C07210=1038.380,356.287,-127.366,172.660,43.947,158.571
C07211=1038.387,356.534,-127.405,172.666,43.949,158.572
C07212=1038.395,356.782,-127.444,172.672,43.953,158.573
C07213=1038.402,357.028,-127.482,172.677,43.955,158.575
C07214=1038.410,357.275,-127.521,172.684,43.958,158.576
C07215=1038.418,357.522,-127.559,172.690,43.962,158.577
C07216=1038.426,357.769,-127.598,172.695,43.965,158.578
C07217=1038.434,358.016,-127.636,172.702,43.968,158.580
C07218=1038.442,358.263,-127.674,172.708,43.971,158.581
C07219=1038.450,358.510,-127.713,172.714,43.974,158.582
C07220=1038.458,358.756,-127.751,172.720,43.978,158.584
C07221=1038.466,359.004,-127.790,172.727,43.981,158.585
C07222=1038.472,359.251,-127.829,172.732,43.983,158.586
C07223=1038.481,359.498,-127.867,172.738,43.987,158.587
C07224=1038.489,359.744,-127.907,172.744,43.990,158.589
C07225=1038.497,359.991,-127.945,172.750,43.993,158.590
C07226=1038.505,360.238,-127.984,172.757,43.996,158.591
C07227=1038.513,360.485,-128.022,172.763,44.000,158.593
C07228=1038.521,360.731,-128.061,172.769,44.003,158.594
C07229=1038.528,360.979,-128.100,172.775,44.006,158.595
C07230=1038.536,361.226,-128.139,172.782,44.009,158.597
C07231=1038.544,361.472,-128.178,172.787,44.013,158.598
C07232=1038.552,361.719,-128.216,172.794,44.016,158.599
C07233=1038.561,361.966,-128.256,172.800,44.019,158.601
C07234=1038.568,362.212,-128.295,172.807,44.022,158.602
C07235=1038.576,362.459,-128.334,172.812,44.026,158.603
C07236=1038.588,362.828,-128.393,172.822,44.031,158.605
C07237=1038.599,363.195,-128.451,172.832,44.036,158.608
C07238=1038.612,363.564,-128.509,172.840,44.041,158.610
C07239=1038.623,363.932,-128.568,172.850,44.046,158.612
C07240=1038.631,364.179,-128.607,172.857,44.049,158.613
C07241=1038.639,364.425,-128.646,172.862,44.052,158.614
C07242=1038.647,364.672,-128.686,172.869,44.056,158.616
C07243=1038.655,364.918,-128.725,172.875,44.059,158.617
C07244=1038.663,365.165,-128.765,172.882,44.063,158.619
C07245=1038.671,365.412,-128.804,172.888,44.067,158.620
C07246=1038.678,365.659,-128.844,172.894,44.070,158.621
C07247=1038.687,365.906,-128.883,172.901,44.073,158.623
C07248=1038.695,366.153,-128.923,172.907,44.077,158.624
C07249=1038.703,366.399,-128.962,172.914,44.080,158.626
C07250=1038.712,366.646,-129.002,172.921,44.083,158.627
C07251=1038.719,366.893,-129.041,172.927,44.087,158.629
C07252=1038.728,367.139,-129.081,172.934,44.091,158.630
C07253=1038.735,367.386,-129.121,172.940,44.094,158.632
C07254=1038.744,367.633,-129.160,172.946,44.098,158.633
C07255=1038.752,367.880,-129.200,172.953,44.101,158.634
C07256=1038.760,368.126,-129.239,172.960,44.105,158.636
C07257=1038.768,368.373,-129.280,172.966,44.109,158.637
C07258=1038.777,368.619,-129.319,172.973,44.112,158.639
C07259=1038.784,368.866,-129.359,172.980,44.115,158.640
C07260=1038.793,369.113,-129.399,172.986,44.119,158.642
C07261=1038.800,369.360,-129.438,172.993,44.123,158.643
C07262=1038.809,369.606,-129.478,172.999,44.126,158.645
C07263=1038.818,369.852,-129.518,173.006,44.130,158.646
C07264=1038.825,370.099,-129.558,173.012,44.134,158.648
C07265=1038.833,370.345,-129.598,173.019,44.137,158.649
C07266=1038.842,370.593,-129.638,173.026,44.141,158.651
C07267=1038.850,370.840,-129.678,173.033,44.145,158.652
C07268=1038.858,371.086,-129.719,173.039,44.149,158.654
C07269=1038.866,371.332,-129.759,173.046,44.152,158.655
C07270=1038.875,371.579,-129.799,173.053,44.156,158.657
C07271=1038.883,371.825,-129.839,173.060,44.159,158.658
C07272=1038.890,372.072,-129.879,173.066,44.163,158.660
C07273=1038.899,372.319,-129.920,173.073,44.168,158.662
C07274=1038.907,372.565,-129.961,173.080,44.171,158.663
C07275=1038.916,372.812,-130.000,173.087,44.175,158.665
C07276=1038.924,373.058,-130.041,173.094,44.179,158.666
C07277=1038.932,373.304,-130.081,173.100,44.182,158.668
C07278=1038.940,373.551,-130.122,173.108,44.187,158.669
C07279=1038.948,373.798,-130.162,173.115,44.190,158.671
C07280=1038.957,374.044,-130.202,173.121,44.194,158.672
C07281=1038.965,374.291,-130.243,173.128,44.198,158.674
C07282=1038.973,374.538,-130.284,173.136,44.202,158.676
C07283=1038.981,374.784,-130.325,173.143,44.206,158.677
C07284=1038.990,375.031,-130.366,173.150,44.210,158.679
C07285=1038.998,375.277,-130.406,173.156,44.214,158.680
C07286=1039.007,375.523,-130.446,173.163,44.217,158.682
C07287=1039.015,375.770,-130.487,173.170,44.221,158.684
C07288=1039.023,376.016,-130.528,173.177,44.225,158.685
C07289=1039.032,376.263,-130.569,173.184,44.229,158.687
C07290=1039.040,376.510,-130.610,173.191,44.233,158.688
C07291=1039.049,376.756,-130.650,173.199,44.237,158.690
C07292=1039.062,377.144,-130.714,173.210,44.244,158.693
C07293=1039.076,377.532,-130.778,173.221,44.250,158.695
C07294=1039.089,377.920,-130.843,173.233,44.256,158.698
C07295=1039.103,378.308,-130.908,173.244,44.263,158.701
C07296=1039.111,378.555,-130.949,173.251,44.266,158.702
C07297=1039.119,378.802,-130.989,173.259,44.270,158.704
C07298=1039.128,379.048,-131.031,173.266,44.275,158.706
C07299=1039.136,379.295,-131.072,173.273,44.279,158.707
C07300=1039.145,379.541,-131.114,173.280,44.283,158.709
C07301=1039.153,379.787,-131.155,173.288,44.287,158.711
C07302=1039.161,380.034,-131.196,173.295,44.291,158.712
C07303=1039.170,380.280,-131.238,173.302,44.296,158.714
C07304=1039.178,380.526,-131.279,173.309,44.300,158.716
C07305=1039.187,380.773,-131.321,173.317,44.304,158.718
C07306=1039.195,381.018,-131.362,173.324,44.308,158.719
C07307=1039.204,381.265,-131.403,173.331,44.312,158.721
C07308=1039.213,381.512,-131.445,173.339,44.317,158.723
C07309=1039.221,381.758,-131.486,173.346,44.321,158.725
C07310=1039.230,382.004,-131.528,173.354,44.325,158.726
C07311=1039.238,382.251,-131.570,173.361,44.329,158.728
C07312=1039.247,382.498,-131.611,173.369,44.334,158.730
C07313=1039.255,382.743,-131.653,173.376,44.338,158.732
C07314=1039.264,382.990,-131.695,173.383,44.343,158.733
C07315=1039.273,383.236,-131.736,173.391,44.347,158.735
C07316=1039.281,383.483,-131.779,173.399,44.351,158.737
C07317=1039.289,383.728,-131.820,173.406,44.355,158.739
C07318=1039.298,383.975,-131.862,173.414,44.360,158.741
C07319=1039.307,384.221,-131.903,173.421,44.364,158.742
C07320=1039.316,384.467,-131.945,173.429,44.369,158.744
C07321=1039.325,384.713,-131.988,173.437,44.373,158.746
C07322=1039.334,384.960,-132.030,173.445,44.378,158.748
C07323=1039.343,385.206,-132.072,173.452,44.382,158.750
C07324=1039.351,385.453,-132.113,173.460,44.387,158.752
C07325=1039.360,385.699,-132.155,173.468,44.391,158.754
C07326=1039.368,385.944,-132.198,173.475,44.395,158.755
C07327=1039.377,386.191,-132.239,173.483,44.400,158.757
C07328=1039.386,386.437,-132.281,173.491,44.405,158.759
C07329=1039.395,386.683,-132.323,173.498,44.409,158.761
C07330=1039.404,386.929,-132.366,173.506,44.414,158.763
C07331=1039.413,387.176,-132.408,173.515,44.418,158.765
C07332=1039.422,387.422,-132.450,173.522,44.423,158.767
C07333=1039.431,387.669,-132.492,173.531,44.427,158.769
C07334=1039.440,387.915,-132.535,173.538,44.432,158.770
C07335=1039.449,388.161,-132.577,173.546,44.437,158.772
C07336=1039.458,388.407,-132.619,173.554,44.441,158.774
C07337=1039.466,388.653,-132.662,173.562,44.446,158.776
C07338=1039.476,388.899,-132.705,173.570,44.450,158.778
C07339=1039.484,389.145,-132.747,173.578,44.455,158.780
C07340=1039.493,389.391,-132.789,173.585,44.460,158.782
C07341=1039.502,389.638,-132.833,173.594,44.464,158.784
C07342=1039.512,389.883,-132.875,173.601,44.469,158.786
C07343=1039.520,390.129,-132.918,173.610,44.474,158.788
C07344=1039.529,390.376,-132.960,173.618,44.479,158.790
C07345=1039.537,390.622,-133.003,173.626,44.483,158.792
C07346=1039.547,390.868,-133.046,173.634,44.489,158.794
C07347=1039.556,391.114,-133.089,173.643,44.493,158.796
C07348=1039.565,391.352,-133.130,173.650,44.498,158.798
C07349=1039.573,391.589,-133.172,173.658,44.502,158.800
C07350=1039.582,391.827,-133.214,173.666,44.507,158.802
C07351=1039.591,392.065,-133.255,173.674,44.512,158.804
C07352=1039.599,392.303,-133.297,173.682,44.517,158.806
C07353=1039.608,392.541,-133.338,173.690,44.521,158.808
C07354=1039.617,392.779,-133.380,173.698,44.526,158.809
C07355=1039.626,393.017,-133.422,173.707,44.531,158.812
C07356=1039.634,393.263,-133.465,173.714,44.536,158.813
C07357=1039.643,393.510,-133.508,173.723,44.541,158.816
C07358=1039.653,393.755,-133.551,173.732,44.546,158.818
C07359=1039.662,394.001,-133.595,173.740,44.551,158.820
C07360=1039.671,394.247,-133.638,173.748,44.555,158.822
C07361=1039.681,394.493,-133.681,173.756,44.561,158.824
C07362=1039.689,394.739,-133.725,173.765,44.566,158.826
C07363=1039.699,394.986,-133.768,173.774,44.571,158.828
C07364=1039.708,395.231,-133.812,173.783,44.576,158.830
C07365=1039.717,395.477,-133.855,173.790,44.581,158.832
C07366=1039.726,395.723,-133.899,173.799,44.586,158.834
C07367=1039.735,395.969,-133.943,173.808,44.591,158.837
C07368=1039.744,396.214,-133.987,173.816,44.596,158.839
C07369=1039.754,396.461,-134.029,173.825,44.602,158.841
C07370=1039.763,396.706,-134.073,173.834,44.607,158.843
C07371=1039.772,396.952,-134.117,173.843,44.612,158.845
C07372=1039.781,397.198,-134.161,173.851,44.617,158.847
C07373=1039.790,397.444,-134.205,173.860,44.623,158.850
C07374=1039.800,397.690,-134.249,173.868,44.628,158.852
C07375=1039.809,397.936,-134.293,173.877,44.632,158.854
C07376=1039.819,398.181,-134.336,173.886,44.638,158.856
C07377=1039.828,398.427,-134.381,173.894,44.643,158.858
C07378=1039.837,398.673,-134.424,173.903,44.649,158.861
C07379=1039.846,398.919,-134.468,173.912,44.654,158.863
C07380=1039.856,399.165,-134.512,173.921,44.659,158.865
C07381=1039.865,399.411,-134.557,173.930,44.664,158.867
C07382=1039.875,399.657,-134.601,173.939,44.670,158.870
C07383=1039.884,399.903,-134.646,173.948,44.675,158.872
C07384=1039.893,400.148,-134.689,173.957,44.680,158.874
C07385=1039.903,400.395,-134.733,173.966,44.686,158.876
C07386=1039.912,400.640,-134.778,173.975,44.691,158.879
C07387=1039.922,400.886,-134.822,173.985,44.697,158.881
C07388=1039.931,401.132,-134.867,173.994,44.702,158.883
C07389=1039.941,401.378,-134.911,174.003,44.708,158.886
C07390=1039.951,401.623,-134.956,174.012,44.714,158.888
C07391=1039.960,401.869,-135.000,174.021,44.719,158.890
C07392=1039.970,402.115,-135.045,174.030,44.725,158.893
C07393=1039.979,402.361,-135.090,174.039,44.730,158.895
C07394=1039.989,402.607,-135.134,174.049,44.736,158.897
C07395=1039.999,402.852,-135.179,174.058,44.741,158.900
C07396=1040.008,403.098,-135.224,174.067,44.747,158.902
C07397=1040.017,403.344,-135.268,174.076,44.753,158.905
C07398=1040.027,403.590,-135.313,174.085,44.758,158.907
C07399=1040.036,403.835,-135.358,174.094,44.764,158.909
C07400=1040.045,404.054,-135.398,174.103,44.769,158.911
C07401=1040.053,404.274,-135.439,174.111,44.774,158.914
C07402=1040.062,404.493,-135.479,174.119,44.779,158.916
C07403=1040.071,404.711,-135.519,174.128,44.784,158.918
C07404=1040.079,404.930,-135.559,174.136,44.789,158.920
C07405=1040.088,405.150,-135.600,174.145,44.794,158.922
C07406=1040.096,405.369,-135.640,174.153,44.800,158.924
C07407=1040.105,405.588,-135.681,174.162,44.805,158.927
C07408=1040.114,405.809,-135.721,174.171,44.810,158.929
C07409=1040.122,406.030,-135.762,174.179,44.816,158.931
C07410=1040.131,406.251,-135.802,174.188,44.820,158.933
C07411=1040.140,406.473,-135.843,174.196,44.826,158.936
C07412=1040.149,406.693,-135.883,174.205,44.831,158.938
C07413=1040.158,406.914,-135.925,174.214,44.837,158.940
C07414=1040.166,407.136,-135.966,174.222,44.842,158.942
C07415=1040.175,407.356,-136.006,174.231,44.847,158.945
C07416=1040.185,407.602,-136.053,174.241,44.853,158.947
C07417=1040.195,407.848,-136.098,174.251,44.859,158.950
C07418=1040.205,408.093,-136.144,174.261,44.865,158.952
C07419=1040.214,408.339,-136.189,174.271,44.871,158.955
C07420=1040.225,408.585,-136.235,174.280,44.877,158.957
C07421=1040.235,408.830,-136.280,174.290,44.883,158.960
C07422=1040.244,409.076,-136.326,174.301,44.889,158.963
C07423=1040.254,409.321,-136.372,174.310,44.895,158.965
C07424=1040.265,409.567,-136.417,174.321,44.901,158.968
C07425=1040.274,409.812,-136.463,174.330,44.907,158.970
C07426=1040.285,410.058,-136.509,174.341,44.913,158.973
C07427=1040.295,410.304,-136.555,174.350,44.920,158.976
C07428=1040.305,410.549,-136.601,174.361,44.925,158.978
C07429=1040.315,410.794,-136.647,174.371,44.932,158.981
C07430=1040.325,411.040,-136.693,174.381,44.938,158.984
C07431=1040.335,411.285,-136.739,174.391,44.944,158.986
C07432=1040.345,411.531,-136.785,174.401,44.950,158.989
C07433=1040.356,411.777,-136.831,174.412,44.957,158.992
C07434=1040.366,412.023,-136.878,174.422,44.963,158.994
C07435=1040.376,412.268,-136.924,174.432,44.969,158.997
C07436=1040.386,412.513,-136.971,174.442,44.976,159.000
C07437=1040.396,412.759,-137.017,174.453,44.982,159.003
C07438=1040.406,413.004,-137.063,174.464,44.988,159.005
C07439=1040.416,413.250,-137.110,174.473,44.995,159.008
C07440=1040.426,413.496,-137.157,174.484,45.001,159.011
C07441=1040.437,413.741,-137.204,174.495,45.008,159.014
C07442=1040.447,413.986,-137.250,174.506,45.014,159.017
C07443=1040.457,414.232,-137.297,174.516,45.020,159.019
C07444=1040.467,414.478,-137.344,174.527,45.027,159.022
C07445=1040.478,414.723,-137.390,174.537,45.034,159.025
C07446=1040.488,414.968,-137.437,174.548,45.040,159.028
C07447=1040.498,415.214,-137.484,174.558,45.047,159.031
C07448=1040.508,415.459,-137.531,174.569,45.053,159.033
C07449=1040.519,415.704,-137.578,174.580,45.060,159.036
C07450=1040.530,415.949,-137.625,174.591,45.067,159.039
C07451=1040.540,416.195,-137.672,174.602,45.073,159.042
C07452=1040.551,416.440,-137.719,174.613,45.080,159.045
C07453=1040.561,416.685,-137.766,174.624,45.086,159.048
C07454=1040.571,416.930,-137.813,174.635,45.093,159.051
C07455=1040.582,417.176,-137.861,174.646,45.099,159.054
C07456=1040.593,417.421,-137.907,174.657,45.106,159.057
C07457=1040.603,417.666,-137.955,174.668,45.113,159.060
C07458=1040.614,417.912,-138.002,174.679,45.120,159.063
C07459=1040.624,418.158,-138.049,174.690,45.127,159.066
C07460=1040.634,418.402,-138.097,174.701,45.134,159.069
C07461=1040.645,418.648,-138.145,174.712,45.141,159.072
C07462=1040.655,418.894,-138.192,174.723,45.147,159.075
C07463=1040.666,419.138,-138.240,174.735,45.154,159.078
C07464=1040.677,419.384,-138.288,174.746,45.161,159.081
C07465=1040.687,419.629,-138.336,174.757,45.168,159.084
C07466=1040.698,419.874,-138.384,174.769,45.175,159.087
C07467=1040.708,420.120,-138.431,174.780,45.182,159.090
C07468=1040.718,420.345,-138.475,174.790,45.189,159.093
C07469=1040.728,420.569,-138.519,174.801,45.195,159.096
C07470=1040.738,420.795,-138.563,174.812,45.201,159.099
C07471=1040.748,421.020,-138.607,174.822,45.208,159.102
C07472=1040.758,421.246,-138.651,174.833,45.214,159.104
C07473=1040.768,421.470,-138.696,174.844,45.221,159.107
C07474=1040.777,421.695,-138.739,174.855,45.227,159.110
C07475=1040.788,421.921,-138.784,174.865,45.234,159.113
C07476=1040.798,422.165,-138.832,174.877,45.241,159.116
C07477=1040.810,422.411,-138.881,174.889,45.248,159.119
C07478=1040.821,422.656,-138.929,174.900,45.255,159.123
C07479=1040.831,422.901,-138.977,174.913,45.262,159.126
C07480=1040.842,423.146,-139.025,174.924,45.270,159.129
C07481=1040.853,423.391,-139.073,174.937,45.277,159.132
C07482=1040.865,423.636,-139.122,174.948,45.284,159.136
C07483=1040.876,423.881,-139.171,174.961,45.292,159.139
C07484=1040.887,424.127,-139.219,174.972,45.299,159.142
C07485=1040.897,424.371,-139.268,174.985,45.307,159.146
C07486=1040.908,424.616,-139.317,174.997,45.314,159.149
C07487=1040.920,424.861,-139.366,175.009,45.321,159.152
C07488=1040.931,425.107,-139.414,175.021,45.329,159.156
C07489=1040.941,425.352,-139.463,175.033,45.336,159.159
C07490=1040.953,425.596,-139.512,175.046,45.344,159.162
C07491=1040.964,425.841,-139.561,175.058,45.351,159.166
C07492=1040.975,426.086,-139.610,175.070,45.359,159.169
C07493=1040.986,426.332,-139.659,175.083,45.366,159.172
C07494=1040.997,426.576,-139.708,175.095,45.374,159.176
C07495=1041.009,426.821,-139.757,175.108,45.381,159.179
C07496=1041.020,427.066,-139.806,175.120,45.389,159.183
C07497=1041.031,427.311,-139.856,175.133,45.397,159.186
C07498=1041.042,427.556,-139.905,175.146,45.404,159.190
C07499=1041.054,427.800,-139.954,175.158,45.412,159.193
C07500=1041.065,428.046,-140.004,175.171,45.420,159.197
C07501=1041.077,428.290,-140.054,175.184,45.427,159.200
C07502=1041.088,428.535,-140.103,175.197,45.435,159.204
C07503=1041.099,428.780,-140.152,175.210,45.443,159.207
C07504=1041.111,429.025,-140.202,175.223,45.451,159.211
C07505=1041.122,429.270,-140.252,175.236,45.458,159.214
C07506=1041.133,429.514,-140.302,175.249,45.466,159.218
C07507=1041.144,429.758,-140.352,175.262,45.474,159.222
C07508=1041.156,430.004,-140.401,175.275,45.482,159.225
C07509=1041.167,430.248,-140.452,175.288,45.490,159.229
C07510=1041.179,430.492,-140.502,175.301,45.498,159.232
C07511=1041.191,430.738,-140.552,175.314,45.506,159.236
C07512=1041.201,430.983,-140.602,175.327,45.515,159.240
C07513=1041.214,431.227,-140.652,175.340,45.523,159.243
C07514=1041.225,431.472,-140.702,175.354,45.530,159.247
C07515=1041.237,431.717,-140.752,175.368,45.539,159.251
C07516=1041.248,431.961,-140.803,175.381,45.547,159.255
C07517=1041.260,432.206,-140.853,175.394,45.555,159.258
C07518=1041.272,432.450,-140.904,175.408,45.563,159.262
C07519=1041.284,432.695,-140.954,175.421,45.571,159.266
C07520=1041.295,432.940,-141.005,175.435,45.579,159.270
C07521=1041.308,433.185,-141.055,175.449,45.588,159.274
C07522=1041.319,433.428,-141.106,175.463,45.596,159.277
C07523=1041.331,433.673,-141.156,175.477,45.604,159.281
C07524=1041.343,433.918,-141.207,175.490,45.613,159.285
C07525=1041.355,434.162,-141.257,175.505,45.621,159.289
C07526=1041.367,434.406,-141.308,175.518,45.629,159.293
C07527=1041.379,434.651,-141.358,175.532,45.637,159.297
C07528=1041.391,434.884,-141.407,175.546,45.646,159.301
C07529=1041.402,435.117,-141.456,175.559,45.653,159.304
C07530=1041.414,435.351,-141.504,175.572,45.662,159.308
C07531=1041.425,435.583,-141.553,175.586,45.669,159.312
C07532=1041.437,435.816,-141.602,175.600,45.678,159.316
C07533=1041.448,436.049,-141.650,175.613,45.686,159.319
C07534=1041.459,436.282,-141.700,175.628,45.694,159.323
C07535=1041.471,436.515,-141.749,175.641,45.702,159.327
C07536=1041.483,436.759,-141.800,175.656,45.711,159.331
C07537=1041.495,437.004,-141.851,175.670,45.720,159.335
C07538=1041.508,437.248,-141.903,175.684,45.728,159.339
C07539=1041.519,437.492,-141.955,175.699,45.737,159.344
C07540=1041.532,437.736,-142.006,175.714,45.746,159.348
C07541=1041.544,437.980,-142.058,175.728,45.754,159.352
C07542=1041.556,438.225,-142.109,175.743,45.763,159.356
C07543=1041.569,438.469,-142.162,175.758,45.772,159.360
C07544=1041.581,438.713,-142.214,175.773,45.781,159.364
C07545=1041.593,438.958,-142.265,175.788,45.789,159.368
C07546=1041.606,439.202,-142.318,175.803,45.799,159.373
C07547=1041.619,439.446,-142.369,175.818,45.808,159.377
C07548=1041.631,439.690,-142.421,175.833,45.817,159.381
C07549=1041.644,439.934,-142.474,175.849,45.825,159.386
C07550=1041.656,440.178,-142.526,175.864,45.834,159.390
C07551=1041.669,440.423,-142.578,175.879,45.844,159.394
C07552=1041.681,440.667,-142.630,175.894,45.853,159.399
C07553=1041.694,440.911,-142.683,175.910,45.861,159.403
C07554=1041.706,441.155,-142.735,175.925,45.871,159.407
C07555=1041.719,441.400,-142.788,175.941,45.880,159.412
C07556=1041.731,441.643,-142.840,175.957,45.889,159.416
C07557=1041.744,441.888,-142.893,175.972,45.898,159.421
C07558=1041.757,442.132,-142.946,175.988,45.907,159.425
C07559=1041.769,442.376,-142.998,176.004,45.917,159.430
C07560=1041.782,442.620,-143.051,176.020,45.926,159.434
C07561=1041.795,442.864,-143.104,176.035,45.935,159.439
C07562=1041.808,443.108,-143.157,176.052,45.944,159.443
C07563=1041.821,443.352,-143.210,176.067,45.954,159.448
C07564=1041.834,443.595,-143.263,176.084,45.964,159.452
C07565=1041.846,443.840,-143.316,176.100,45.973,159.457
C07566=1041.860,444.084,-143.369,176.116,45.982,159.461
C07567=1041.873,444.328,-143.422,176.132,45.992,159.466
C07568=1041.886,444.570,-143.475,176.149,46.001,159.471
C07569=1041.899,444.814,-143.528,176.165,46.011,159.476
C07570=1041.913,445.057,-143.581,176.182,46.020,159.480
C07571=1041.927,445.301,-143.634,176.199,46.030,159.485
C07572=1041.941,445.544,-143.686,176.215,46.039,159.489
C07573=1041.957,445.787,-143.737,176.231,46.048,159.494
C07574=1041.972,446.031,-143.788,176.248,46.057,159.499
C07575=1041.989,446.275,-143.839,176.265,46.066,159.503
C07576=1042.006,446.519,-143.889,176.282,46.075,159.508
C07577=1042.023,446.762,-143.939,176.299,46.083,159.512
C07578=1042.042,447.006,-143.988,176.316,46.092,159.517
C07579=1042.060,447.251,-144.037,176.333,46.100,159.521
C07580=1042.080,447.495,-144.084,176.351,46.109,159.526
C07581=1042.100,447.740,-144.132,176.368,46.117,159.530
C07582=1042.120,447.984,-144.180,176.385,46.125,159.535
C07583=1042.141,448.229,-144.226,176.402,46.133,159.539
C07584=1042.163,448.473,-144.273,176.420,46.141,159.544
C07585=1042.186,448.718,-144.319,176.439,46.149,159.548
C07586=1042.209,448.963,-144.364,176.455,46.157,159.552
C07587=1042.232,449.208,-144.408,176.473,46.165,159.557
C07588=1042.264,449.526,-144.466,176.497,46.174,159.562
C07589=1042.296,449.843,-144.523,176.520,46.184,159.568
C07590=1042.330,450.161,-144.579,176.543,46.193,159.573
C07591=1042.365,450.479,-144.633,176.567,46.202,159.579
C07592=1042.392,450.725,-144.676,176.586,46.209,159.583
C07593=1042.420,450.970,-144.717,176.603,46.216,159.587
C07594=1042.448,451.215,-144.758,176.622,46.223,159.592
C07595=1042.477,451.461,-144.799,176.641,46.230,159.596
C07596=1042.177,451.505,-145.113,176.644,46.308,159.620
C07597=1042.148,451.260,-145.073,176.625,46.302,159.616
C07598=1042.119,451.014,-145.032,176.606,46.295,159.611
C07599=1042.091,450.768,-144.991,176.588,46.289,159.607
C07600=1042.064,450.523,-144.949,176.570,46.281,159.603
C07601=1042.031,450.221,-144.897,176.546,46.273,159.598
C07602=1041.999,449.918,-144.844,176.524,46.264,159.592
C07603=1041.968,449.615,-144.790,176.502,46.255,159.587
C07604=1041.937,449.314,-144.736,176.480,46.246,159.582
C07605=1041.913,449.069,-144.692,176.462,46.238,159.577
C07606=1041.890,448.824,-144.646,176.444,46.231,159.573
C07607=1041.867,448.578,-144.600,176.427,46.223,159.568
C07608=1041.845,448.334,-144.555,176.409,46.215,159.564
C07609=1041.823,448.090,-144.508,176.391,46.207,159.560
C07610=1041.803,447.845,-144.461,176.373,46.199,159.555
C07611=1041.782,447.601,-144.414,176.356,46.191,159.551
C07612=1041.762,447.356,-144.366,176.339,46.183,159.546
C07613=1041.743,447.111,-144.317,176.321,46.174,159.542
C07614=1041.724,446.868,-144.268,176.304,46.166,159.537
C07615=1041.706,446.624,-144.219,176.287,46.157,159.533
C07616=1041.689,446.381,-144.169,176.270,46.149,159.528
C07617=1041.672,446.136,-144.118,176.253,46.140,159.524
C07618=1041.657,445.892,-144.068,176.236,46.131,159.519
C07619=1041.641,445.649,-144.016,176.219,46.122,159.514
C07620=1041.625,445.406,-143.965,176.203,46.113,159.510
C07621=1041.612,445.161,-143.913,176.186,46.104,159.505
C07622=1041.597,444.919,-143.860,176.170,46.095,159.501
C07623=1041.585,444.675,-143.807,176.153,46.085,159.496
C07624=1041.571,444.433,-143.755,176.137,46.076,159.491
C07625=1041.558,444.189,-143.701,176.120,46.067,159.487
C07626=1041.545,443.945,-143.648,176.103,46.057,159.482
C07627=1041.532,443.701,-143.595,176.088,46.048,159.477
C07628=1041.519,443.457,-143.542,176.072,46.038,159.473
C07629=1041.505,443.213,-143.489,176.055,46.029,159.468
C07630=1041.493,442.969,-143.436,176.040,46.020,159.464
C07631=1041.480,442.725,-143.383,176.023,46.011,159.459
C07632=1041.467,442.481,-143.330,176.007,46.001,159.455
C07633=1041.454,442.237,-143.277,175.992,45.992,159.450
C07634=1041.441,441.993,-143.224,175.975,45.983,159.446
C07635=1041.429,441.749,-143.172,175.960,45.974,159.441
C07636=1041.416,441.505,-143.119,175.944,45.965,159.437
C07637=1041.403,441.260,-143.066,175.928,45.955,159.432
C07638=1041.391,441.017,-143.014,175.913,45.946,159.428
C07639=1041.378,440.773,-142.961,175.897,45.938,159.424
C07640=1041.366,440.529,-142.909,175.882,45.929,159.419
C07641=1041.353,440.284,-142.857,175.867,45.920,159.415
C07642=1041.341,440.040,-142.804,175.851,45.911,159.411
C07643=1041.328,439.796,-142.752,175.836,45.902,159.406
C07644=1041.316,439.552,-142.700,175.821,45.893,159.402
C07645=1041.302,439.307,-142.648,175.806,45.884,159.398
C07646=1041.290,439.063,-142.597,175.791,45.875,159.393
C07647=1041.278,438.819,-142.544,175.775,45.866,159.389
C07648=1041.265,438.574,-142.492,175.760,45.858,159.385
C07649=1041.253,438.330,-142.441,175.745,45.849,159.381
C07650=1041.241,438.086,-142.388,175.730,45.840,159.377
C07651=1041.229,437.842,-142.337,175.715,45.832,159.373
C07652=1041.216,437.598,-142.285,175.700,45.823,159.368
C07653=1041.204,437.353,-142.234,175.686,45.814,159.364
C07654=1041.192,437.109,-142.182,175.672,45.805,159.360
C07655=1041.180,436.864,-142.130,175.657,45.797,159.356
C07656=1041.167,436.620,-142.079,175.643,45.789,159.352
C07657=1041.156,436.386,-142.030,175.628,45.781,159.348
C07658=1041.144,436.152,-141.981,175.615,45.772,159.344
C07659=1041.133,435.919,-141.932,175.601,45.764,159.340
C07660=1041.121,435.685,-141.883,175.587,45.756,159.336
C07661=1041.110,435.452,-141.834,175.574,45.748,159.333
C07662=1041.099,435.218,-141.785,175.560,45.740,159.329
C07663=1041.087,434.985,-141.736,175.546,45.732,159.325
C07664=1041.075,434.751,-141.688,175.533,45.724,159.321
C07665=1041.064,434.506,-141.637,175.518,45.716,159.317
C07666=1041.051,434.262,-141.586,175.505,45.707,159.314
C07667=1041.039,434.017,-141.535,175.491,45.699,159.310
C07668=1041.027,433.773,-141.485,175.477,45.691,159.306
C07669=1041.015,433.528,-141.434,175.463,45.683,159.302
C07670=1041.003,433.284,-141.383,175.449,45.674,159.298
C07671=1040.992,433.039,-141.333,175.435,45.666,159.294
C07672=1040.979,432.794,-141.283,175.422,45.658,159.290
C07673=1040.968,432.550,-141.232,175.407,45.650,159.287
C07674=1040.956,432.305,-141.181,175.394,45.642,159.283
C07675=1040.944,432.060,-141.131,175.381,45.634,159.279
C07676=1040.932,431.816,-141.081,175.367,45.626,159.275
C07677=1040.921,431.571,-141.030,175.353,45.618,159.272
C07678=1040.909,431.327,-140.981,175.340,45.609,159.268
C07679=1040.898,431.082,-140.930,175.327,45.601,159.264
C07680=1040.886,430.838,-140.880,175.313,45.594,159.260
C07681=1040.874,430.593,-140.830,175.300,45.586,159.257
C07682=1040.863,430.348,-140.780,175.287,45.578,159.253
C07683=1040.851,430.103,-140.730,175.274,45.570,159.250
C07684=1040.840,429.859,-140.680,175.261,45.562,159.246
C07685=1040.829,429.614,-140.630,175.248,45.554,159.242
C07686=1040.817,429.369,-140.580,175.235,45.546,159.239
C07687=1040.806,429.124,-140.530,175.221,45.538,159.235
C07688=1040.794,428.880,-140.480,175.209,45.531,159.232
C07689=1040.783,428.634,-140.430,175.196,45.523,159.228
C07690=1040.771,428.390,-140.381,175.183,45.516,159.224
C07691=1040.760,428.145,-140.331,175.170,45.508,159.221
C07692=1040.749,427.900,-140.282,175.157,45.500,159.217
C07693=1040.737,427.656,-140.233,175.144,45.492,159.214
C07694=1040.726,427.410,-140.183,175.131,45.485,159.210
C07695=1040.715,427.165,-140.134,175.119,45.477,159.207
C07696=1040.703,426.920,-140.085,175.106,45.470,159.203
C07697=1040.692,426.676,-140.036,175.093,45.462,159.200
C07698=1040.681,426.431,-139.986,175.081,45.455,159.197
C07699=1040.670,426.186,-139.937,175.069,45.447,159.193
C07700=1040.658,425.941,-139.888,175.056,45.440,159.190
C07701=1040.647,425.696,-139.839,175.043,45.432,159.186
C07702=1040.636,425.451,-139.790,175.031,45.425,159.183
C07703=1040.625,425.206,-139.741,175.019,45.417,159.180
C07704=1040.614,424.961,-139.692,175.006,45.410,159.176
C07705=1040.602,424.717,-139.643,174.995,45.402,159.173
C07706=1040.592,424.471,-139.595,174.982,45.396,159.170
C07707=1040.581,424.227,-139.546,174.969,45.388,159.166
C07708=1040.570,423.982,-139.498,174.958,45.381,159.163
C07709=1040.559,423.737,-139.449,174.945,45.373,159.160
C07710=1040.548,423.491,-139.400,174.934,45.366,159.156
C07711=1040.537,423.246,-139.352,174.921,45.359,159.153
C07712=1040.526,423.001,-139.304,174.910,45.352,159.150
C07713=1040.515,422.757,-139.255,174.898,45.345,159.147
C07714=1040.504,422.511,-139.207,174.886,45.338,159.144
C07715=1040.493,422.266,-139.158,174.874,45.331,159.140
C07716=1040.482,422.021,-139.110,174.862,45.324,159.137
C07717=1040.472,421.794,-139.065,174.851,45.317,159.134
C07718=1040.462,421.569,-139.021,174.840,45.310,159.131
C07719=1040.452,421.343,-138.977,174.830,45.304,159.128
C07720=1040.442,421.115,-138.933,174.819,45.297,159.125
C07721=1040.432,420.890,-138.889,174.808,45.291,159.123
C07722=1040.422,420.663,-138.844,174.797,45.284,159.120
C07723=1040.411,420.437,-138.800,174.787,45.278,159.117
C07724=1040.402,420.210,-138.756,174.776,45.272,159.114
C07725=1040.392,419.965,-138.708,174.765,45.264,159.111
C07726=1040.381,419.720,-138.659,174.753,45.258,159.108
C07727=1040.370,419.475,-138.612,174.742,45.251,159.105
C07728=1040.359,419.229,-138.564,174.730,45.244,159.102
C07729=1040.349,418.984,-138.517,174.719,45.237,159.099
C07730=1040.339,418.740,-138.469,174.708,45.231,159.096
C07731=1040.328,418.494,-138.421,174.697,45.223,159.093
C07732=1040.318,418.248,-138.374,174.686,45.217,159.090
C07733=1040.307,418.004,-138.326,174.674,45.210,159.087
C07734=1040.296,417.758,-138.278,174.663,45.203,159.084
C07735=1040.285,417.513,-138.232,174.652,45.197,159.081
C07736=1040.275,417.267,-138.185,174.640,45.190,159.078
C07737=1040.264,417.021,-138.137,174.630,45.184,159.075
C07738=1040.254,416.776,-138.090,174.619,45.177,159.072
C07739=1040.243,416.531,-138.043,174.607,45.170,159.069
C07740=1040.233,416.286,-137.996,174.597,45.164,159.066
C07741=1040.223,416.041,-137.949,174.586,45.157,159.063
C07742=1040.212,415.796,-137.902,174.575,45.150,159.060
C07743=1040.201,415.550,-137.854,174.565,45.144,159.057
C07744=1040.191,415.304,-137.807,174.554,45.137,159.054
C07745=1040.181,415.059,-137.760,174.543,45.131,159.052
C07746=1040.170,414.813,-137.714,174.532,45.125,159.049
C07747=1040.160,414.568,-137.667,174.521,45.118,159.046
C07748=1040.150,414.323,-137.620,174.510,45.112,159.043
C07749=1040.139,414.077,-137.574,174.499,45.105,159.040
C07750=1040.129,413.832,-137.527,174.490,45.099,159.038
C07751=1040.120,413.587,-137.480,174.479,45.093,159.035
C07752=1040.109,413.342,-137.434,174.468,45.086,159.032
C07753=1040.099,413.096,-137.387,174.457,45.079,159.029
C07754=1040.089,412.851,-137.340,174.447,45.073,159.026
C07755=1040.079,412.605,-137.294,174.437,45.067,159.024
C07756=1040.068,412.360,-137.247,174.426,45.061,159.021
C07757=1040.059,412.115,-137.201,174.416,45.054,159.018
C07758=1040.049,411.869,-137.154,174.406,45.048,159.015
C07759=1040.038,411.623,-137.108,174.395,45.042,159.013
C07760=1040.028,411.377,-137.062,174.385,45.036,159.010
C07761=1040.018,411.132,-137.016,174.374,45.030,159.007
C07762=1040.008,410.887,-136.970,174.365,45.023,159.005
C07763=1039.998,410.641,-136.924,174.354,45.017,159.002
C07764=1039.987,410.395,-136.878,174.344,45.011,158.999
C07765=1039.977,410.150,-136.832,174.334,45.005,158.997
C07766=1039.967,409.904,-136.786,174.324,44.999,158.994
C07767=1039.957,409.659,-136.740,174.314,44.993,158.991
C07768=1039.947,409.414,-136.695,174.303,44.987,158.989
C07769=1039.937,409.167,-136.649,174.294,44.981,158.986
C07770=1039.926,408.922,-136.603,174.283,44.975,158.984
C07771=1039.917,408.677,-136.557,174.274,44.969,158.981
C07772=1039.907,408.430,-136.512,174.263,44.963,158.978
C07773=1039.897,408.185,-136.466,174.254,44.957,158.976
C07774=1039.887,407.939,-136.420,174.244,44.951,158.973
C07775=1039.877,407.694,-136.375,174.234,44.945,158.971
C07776=1039.867,407.448,-136.330,174.224,44.939,158.968
C07777=1039.858,407.226,-136.288,174.215,44.934,158.966
C07778=1039.849,407.004,-136.247,174.206,44.929,158.964
C07779=1039.840,406.782,-136.206,174.198,44.924,158.962
C07780=1039.831,406.559,-136.165,174.189,44.918,158.959
C07781=1039.823,406.338,-136.124,174.180,44.913,158.957
C07782=1039.814,406.116,-136.083,174.172,44.908,158.955
C07783=1039.805,405.893,-136.042,174.163,44.902,158.952
C07784=1039.796,405.671,-136.001,174.154,44.897,158.950
C07785=1039.787,405.425,-135.955,174.144,44.891,158.948
C07786=1039.777,405.179,-135.911,174.135,44.886,158.945
C07787=1039.767,404.934,-135.866,174.126,44.880,158.943
C07788=1039.758,404.688,-135.820,174.116,44.875,158.940
C07789=1039.749,404.443,-135.775,174.106,44.869,158.938
C07790=1039.738,404.197,-135.730,174.097,44.863,158.936
C07791=1039.729,403.951,-135.685,174.088,44.858,158.933
C07792=1039.720,403.705,-135.640,174.078,44.852,158.931
C07793=1039.710,403.459,-135.595,174.069,44.846,158.928
C07794=1039.700,403.214,-135.550,174.060,44.841,158.926
C07795=1039.691,402.968,-135.505,174.050,44.835,158.924
C07796=1039.681,402.723,-135.460,174.041,44.829,158.921
C07797=1039.672,402.477,-135.416,174.031,44.824,158.919
C07798=1039.662,402.231,-135.371,174.022,44.818,158.916
C07799=1039.653,401.985,-135.326,174.013,44.813,158.914
C07800=1039.643,401.739,-135.282,174.004,44.807,158.912
C07801=1039.633,401.494,-135.237,173.995,44.802,158.909
C07802=1039.624,401.248,-135.193,173.986,44.797,158.907
C07803=1039.614,401.002,-135.149,173.977,44.791,158.905
C07804=1039.605,400.756,-135.104,173.968,44.786,158.903
C07805=1039.595,400.511,-135.060,173.958,44.780,158.900
C07806=1039.586,400.264,-135.016,173.949,44.775,158.898
C07807=1039.576,400.018,-134.971,173.940,44.770,158.896
C07808=1039.567,399.773,-134.927,173.931,44.764,158.893
C07809=1039.558,399.527,-134.883,173.922,44.759,158.891
C07810=1039.548,399.281,-134.839,173.913,44.754,158.889
C07811=1039.539,399.035,-134.795,173.904,44.748,158.887
C07812=1039.529,398.790,-134.750,173.895,44.743,158.884
C07813=1039.520,398.544,-134.706,173.886,44.738,158.882
C07814=1039.511,398.298,-134.662,173.878,44.733,158.880
C07815=1039.501,398.052,-134.618,173.869,44.728,158.878
C07816=1039.492,397.806,-134.574,173.861,44.723,158.876
C07817=1039.483,397.561,-134.531,173.851,44.717,158.873
C07818=1039.473,397.314,-134.486,173.843,44.712,158.871
C07819=1039.464,397.068,-134.442,173.834,44.707,158.869
C07820=1039.455,396.823,-134.399,173.826,44.702,158.867
C07821=1039.446,396.576,-134.355,173.817,44.696,158.865
C07822=1039.436,396.331,-134.312,173.808,44.691,158.862
C07823=1039.427,396.085,-134.268,173.799,44.686,158.860
C07824=1039.418,395.839,-134.224,173.790,44.681,158.858
C07825=1039.409,395.593,-134.181,173.782,44.676,158.856
C07826=1039.400,395.347,-134.137,173.773,44.671,158.854
C07827=1039.390,395.101,-134.094,173.765,44.666,158.852
C07828=1039.381,394.855,-134.050,173.757,44.661,158.850
C07829=1039.372,394.609,-134.006,173.748,44.656,158.848
C07830=1039.362,394.363,-133.964,173.739,44.651,158.846
C07831=1039.354,394.117,-133.920,173.730,44.646,158.843
C07832=1039.345,393.871,-133.877,173.723,44.641,158.841
C07833=1039.334,393.573,-133.824,173.712,44.635,158.839
C07834=1039.323,393.275,-133.772,173.702,44.629,158.836
C07835=1039.312,392.977,-133.720,173.691,44.623,158.834
C07836=1039.300,392.680,-133.667,173.681,44.618,158.831
C07837=1039.287,392.307,-133.602,173.669,44.611,158.828
C07838=1039.273,391.934,-133.536,173.657,44.603,158.825
C07839=1039.259,391.562,-133.472,173.644,44.596,158.822
C07840=1039.246,391.189,-133.407,173.632,44.588,158.819
C07841=1039.237,390.943,-133.364,173.623,44.584,158.817
C07842=1039.228,390.696,-133.320,173.616,44.579,158.815
C07843=1039.219,390.451,-133.278,173.607,44.574,158.813
C07844=1039.210,390.205,-133.235,173.599,44.569,158.811
C07845=1039.201,389.959,-133.192,173.591,44.565,158.809
C07846=1039.192,389.713,-133.151,173.583,44.560,158.807
C07847=1039.183,389.466,-133.107,173.575,44.556,158.805
C07848=1039.174,389.220,-133.065,173.567,44.551,158.803
C07849=1039.165,388.974,-133.022,173.559,44.547,158.801
C07850=1039.156,388.728,-132.979,173.551,44.541,158.799
C07851=1039.148,388.482,-132.937,173.542,44.537,158.797
C07852=1039.139,388.236,-132.895,173.535,44.533,158.796
C07853=1039.130,387.990,-132.852,173.526,44.528,158.794
C07854=1039.121,387.743,-132.810,173.519,44.523,158.792
C07855=1039.112,387.498,-132.767,173.511,44.519,158.790
C07856=1039.103,387.250,-132.725,173.503,44.514,158.788
C07857=1039.094,387.005,-132.682,173.495,44.510,158.786
C07858=1039.085,386.758,-132.641,173.487,44.506,158.784
C07859=1039.076,386.512,-132.599,173.479,44.501,158.782
C07860=1039.067,386.266,-132.556,173.472,44.496,158.780
C07861=1039.059,386.019,-132.514,173.463,44.492,158.779
C07862=1039.050,385.773,-132.472,173.456,44.488,158.777
C07863=1039.040,385.527,-132.430,173.448,44.483,158.775
C07864=1039.031,385.281,-132.388,173.440,44.479,158.773
C07865=1039.023,385.035,-132.347,173.432,44.474,158.771
C07866=1039.015,384.789,-132.305,173.425,44.470,158.769
C07867=1039.006,384.542,-132.263,173.418,44.466,158.768
C07868=1038.997,384.296,-132.221,173.409,44.461,158.766
C07869=1038.988,384.050,-132.179,173.402,44.457,158.764
C07870=1038.979,383.804,-132.137,173.394,44.452,158.762
C07871=1038.971,383.557,-132.095,173.386,44.449,158.760
C07872=1038.962,383.311,-132.053,173.379,44.444,158.759
C07873=1038.953,383.065,-132.012,173.371,44.440,158.757
C07874=1038.944,382.819,-131.970,173.364,44.435,158.755
C07875=1038.936,382.572,-131.928,173.357,44.431,158.753
C07876=1038.927,382.326,-131.886,173.348,44.427,158.751
C07877=1038.919,382.079,-131.845,173.341,44.423,158.750
C07878=1038.910,381.833,-131.804,173.334,44.418,158.748
C07879=1038.901,381.587,-131.762,173.326,44.414,158.746
C07880=1038.893,381.341,-131.721,173.319,44.410,158.744
C07881=1038.884,381.095,-131.679,173.312,44.406,158.743
C07882=1038.876,380.847,-131.637,173.305,44.402,158.741
C07883=1038.868,380.602,-131.596,173.296,44.398,158.739
C07884=1038.859,380.355,-131.554,173.289,44.394,158.737
C07885=1038.850,380.108,-131.513,173.282,44.389,158.736
C07886=1038.842,379.863,-131.472,173.274,44.385,158.734
C07887=1038.833,379.616,-131.431,173.267,44.381,158.732
C07888=1038.826,379.370,-131.389,173.260,44.377,158.731
C07889=1038.817,379.123,-131.347,173.253,44.373,158.729
C07890=1038.809,378.877,-131.307,173.245,44.368,158.727
C07891=1038.800,378.631,-131.265,173.238,44.365,158.726
C07892=1038.792,378.384,-131.224,173.231,44.361,158.724
C07893=1038.778,377.994,-131.159,173.220,44.354,158.721
C07894=1038.765,377.603,-131.094,173.208,44.348,158.718
C07895=1038.751,377.214,-131.030,173.197,44.342,158.716
C07896=1038.738,376.823,-130.965,173.185,44.335,158.713
C07897=1038.730,376.576,-130.925,173.178,44.332,158.712
C07898=1038.721,376.330,-130.883,173.171,44.327,158.710
C07899=1038.712,376.084,-130.843,173.164,44.324,158.708
C07900=1038.703,375.837,-130.802,173.157,44.320,158.707
C07901=1038.695,375.591,-130.761,173.150,44.316,158.705
C07902=1038.687,375.344,-130.720,173.143,44.312,158.704
C07903=1038.679,375.098,-130.680,173.135,44.308,158.702
C07904=1038.671,374.851,-130.639,173.128,44.304,158.700
C07905=1038.661,374.605,-130.599,173.121,44.301,158.699
C07906=1038.653,374.358,-130.558,173.114,44.297,158.697
C07907=1038.646,374.111,-130.518,173.107,44.293,158.696
C07908=1038.637,373.864,-130.477,173.101,44.289,158.694
C07909=1038.629,373.618,-130.436,173.094,44.285,158.693
C07910=1038.620,373.372,-130.396,173.087,44.282,158.691
C07911=1038.612,373.126,-130.356,173.080,44.278,158.689
C07912=1038.604,372.878,-130.315,173.073,44.274,158.688
C07913=1038.596,372.632,-130.275,173.066,44.270,158.686
C07914=1038.588,372.386,-130.234,173.059,44.267,158.685
C07915=1038.579,372.139,-130.195,173.053,44.263,158.683
C07916=1038.571,371.893,-130.154,173.046,44.259,158.682
C07917=1038.563,371.646,-130.113,173.039,44.255,158.680
C07918=1038.555,371.399,-130.073,173.032,44.252,158.679
C07919=1038.546,371.153,-130.033,173.025,44.248,158.677
C07920=1038.538,370.906,-129.993,173.019,44.244,158.675
C07921=1038.530,370.660,-129.953,173.012,44.241,158.674
C07922=1038.523,370.413,-129.913,173.005,44.237,158.672
C07923=1038.515,370.167,-129.872,172.998,44.233,158.671
C07924=1038.506,369.920,-129.833,172.992,44.229,158.669
C07925=1038.497,369.673,-129.793,172.985,44.226,158.668
C07926=1038.489,369.426,-129.752,172.978,44.223,158.666
C07927=1038.481,369.180,-129.713,172.971,44.219,158.665
C07928=1038.473,368.933,-129.673,172.964,44.215,158.663
C07929=1038.464,368.686,-129.634,172.959,44.212,158.662
C07930=1038.456,368.440,-129.593,172.952,44.208,158.661
C07931=1038.448,368.193,-129.554,172.945,44.205,158.659
C07932=1038.440,367.946,-129.514,172.939,44.201,158.658
C07933=1038.432,367.700,-129.475,172.932,44.198,158.656
C07934=1038.424,367.453,-129.435,172.925,44.195,158.655
C07935=1038.416,367.206,-129.395,172.918,44.191,158.653
C07936=1038.408,366.959,-129.355,172.912,44.188,158.652
C07937=1038.399,366.713,-129.316,172.905,44.184,158.650
C07938=1038.391,366.466,-129.277,172.899,44.181,158.649
C07939=1038.383,366.219,-129.237,172.893,44.177,158.647
C07940=1038.375,365.973,-129.198,172.886,44.174,158.646
C07941=1038.367,365.726,-129.158,172.880,44.171,158.645
C07942=1038.359,365.479,-129.118,172.873,44.167,158.643
C07943=1038.351,365.232,-129.078,172.867,44.164,158.642
C07944=1038.343,364.987,-129.039,172.861,44.160,158.640
C07945=1038.336,364.739,-129.000,172.854,44.157,158.639
C07946=1038.327,364.492,-128.961,172.847,44.154,158.638
C07947=1038.319,364.246,-128.922,172.841,44.150,158.636
C07948=1038.311,363.999,-128.882,172.834,44.147,158.635
C07949=1038.299,363.629,-128.823,172.825,44.142,158.633
C07950=1038.287,363.259,-128.764,172.816,44.137,158.631
C07951=1038.276,362.889,-128.706,172.807,44.132,158.629
C07952=1038.264,362.519,-128.647,172.797,44.127,158.627
C07953=1038.256,362.271,-128.608,172.790,44.124,158.625
C07954=1038.248,362.025,-128.568,172.784,44.120,158.624
C07955=1038.240,361.778,-128.530,172.778,44.117,158.623
C07956=1038.232,361.531,-128.490,172.772,44.114,158.621
C07957=1038.224,361.284,-128.451,172.765,44.111,158.620
C07958=1038.216,361.037,-128.413,172.760,44.108,158.619
C07959=1038.208,360.791,-128.374,172.753,44.104,158.617
C07960=1038.200,360.544,-128.335,172.747,44.101,158.616
C07961=1038.192,360.297,-128.297,172.740,44.098,158.615
C07962=1038.185,360.050,-128.257,172.735,44.095,158.613
C07963=1038.177,359.803,-128.218,172.728,44.091,158.612
C07964=1038.169,359.556,-128.180,172.722,44.089,158.611
C07965=1038.161,359.309,-128.142,172.716,44.086,158.609
C07966=1038.152,359.063,-128.102,172.710,44.082,158.608
C07967=1038.145,358.816,-128.064,172.704,44.079,158.607
C07968=1038.137,358.569,-128.025,172.698,44.076,158.606
C07969=1038.129,358.322,-127.987,172.692,44.073,158.604
C07970=1038.121,358.075,-127.949,172.685,44.070,158.603
C07971=1038.114,357.828,-127.909,172.680,44.067,158.602
C07972=1038.106,357.581,-127.871,172.673,44.064,158.600
C07973=1038.098,357.334,-127.833,172.667,44.061,158.599
C07974=1038.090,357.088,-127.794,172.662,44.058,158.598
C07975=1038.082,356.840,-127.756,172.655,44.055,158.597
C07976=1038.075,356.594,-127.717,172.650,44.051,158.595
C07977=1038.067,356.347,-127.679,172.644,44.049,158.594
C07978=1038.059,356.100,-127.641,172.637,44.046,158.593
C07979=1038.051,355.853,-127.602,172.632,44.043,158.592
C07980=1038.044,355.606,-127.564,172.625,44.040,158.590
C07981=1038.035,355.359,-127.526,172.620,44.037,158.589
C07982=1038.028,355.112,-127.488,172.614,44.034,158.588
C07983=1038.020,354.865,-127.449,172.608,44.031,158.587
C07984=1038.012,354.618,-127.412,172.602,44.028,158.585
C07985=1038.004,354.371,-127.374,172.596,44.025,158.584
C07986=1037.996,354.124,-127.335,172.590,44.022,158.583
C07987=1037.989,353.877,-127.298,172.584,44.020,158.582
C07988=1037.981,353.630,-127.259,172.579,44.016,158.581
C07989=1037.973,353.383,-127.221,172.572,44.014,158.579
C07990=1037.966,353.136,-127.183,172.567,44.011,158.578
C07991=1037.958,352.889,-127.145,172.561,44.008,158.577
C07992=1037.950,352.642,-127.108,172.555,44.005,158.576
C07993=1037.942,352.396,-127.070,172.549,44.002,158.575
C07994=1037.934,352.148,-127.032,172.544,43.999,158.573
C07995=1037.927,351.901,-126.993,172.538,43.996,158.572
C07996=1037.920,351.654,-126.956,172.532,43.994,158.571
C07997=1037.912,351.408,-126.918,172.526,43.991,158.570
C07998=1037.904,351.160,-126.880,172.521,43.988,158.569
C07999=1037.897,350.913,-126.842,172.515,43.985,158.567
C08000=1037.889,350.667,-126.805,172.509,43.983,158.566
C08001=1037.881,350.419,-126.767,172.503,43.980,158.565
C08002=1037.874,350.172,-126.729,172.498,43.977,158.564
C08003=1037.866,349.925,-126.691,172.492,43.974,158.563
C08004=1037.859,349.678,-126.653,172.487,43.971,158.562
C08005=1037.847,349.314,-126.598,172.478,43.968,158.560
C08006=1037.836,348.950,-126.543,172.470,43.963,158.558
C08007=1037.825,348.586,-126.488,172.461,43.959,158.557
C08008=1037.814,348.221,-126.432,172.453,43.955,158.555
C08009=1037.806,347.974,-126.395,172.448,43.953,158.554
C08010=1037.798,347.727,-126.358,172.442,43.950,158.553
C08011=1037.790,347.480,-126.321,172.436,43.948,158.552
C08012=1037.783,347.233,-126.283,172.431,43.945,158.550
C08013=1037.776,346.986,-126.246,172.425,43.942,158.549
C08014=1037.768,346.739,-126.209,172.420,43.939,158.548
C08015=1037.761,346.492,-126.171,172.415,43.937,158.547
C08016=1037.753,346.245,-126.134,172.409,43.934,158.546
C08017=1037.745,345.998,-126.097,172.403,43.932,158.545
C08018=1037.738,345.751,-126.059,172.397,43.929,158.544
C08019=1037.730,345.504,-126.022,172.392,43.927,158.543
C08020=1037.723,345.256,-125.985,172.387,43.924,158.542
C08021=1037.715,345.009,-125.948,172.381,43.921,158.540
C08022=1037.707,344.762,-125.911,172.376,43.919,158.539
C08023=1037.699,344.515,-125.874,172.370,43.916,158.538
C08024=1037.692,344.267,-125.837,172.365,43.914,158.537
C08025=1037.684,344.020,-125.800,172.360,43.911,158.536
C08026=1037.677,343.773,-125.763,172.354,43.908,158.535
C08027=1037.670,343.527,-125.726,172.348,43.906,158.534
C08028=1037.663,343.279,-125.689,172.343,43.903,158.533
C08029=1037.655,343.033,-125.652,172.337,43.901,158.532
C08030=1037.648,342.785,-125.616,172.332,43.898,158.531
C08031=1037.640,342.538,-125.579,172.327,43.896,158.530
C08032=1037.633,342.291,-125.541,172.321,43.893,158.529
C08033=1037.625,342.043,-125.505,172.316,43.891,158.528
C08034=1037.618,341.796,-125.467,172.311,43.888,158.527
C08035=1037.610,341.549,-125.431,172.305,43.886,158.526
C08036=1037.603,341.302,-125.394,172.300,43.883,158.525
C08037=1037.596,341.055,-125.358,172.295,43.881,158.524
C08038=1037.588,340.808,-125.322,172.290,43.879,158.523
C08039=1037.580,340.561,-125.285,172.284,43.876,158.521
C08040=1037.573,340.313,-125.248,172.279,43.874,158.520
C08041=1037.566,340.065,-125.212,172.274,43.872,158.519
C08042=1037.558,339.819,-125.175,172.269,43.870,158.519
C08043=1037.550,339.571,-125.138,172.263,43.867,158.517
C08044=1037.544,339.324,-125.102,172.258,43.865,158.516
C08045=1037.536,339.077,-125.066,172.253,43.862,158.515
C08046=1037.528,338.830,-125.029,172.248,43.860,158.514
C08047=1037.520,338.582,-124.993,172.242,43.857,158.513
C08048=1037.513,338.335,-124.956,172.237,43.855,158.512
C08049=1037.506,338.088,-124.920,172.232,43.853,158.511
C08050=1037.499,337.841,-124.884,172.226,43.851,158.510
C08051=1037.491,337.593,-124.847,172.221,43.848,158.509
C08052=1037.485,337.346,-124.811,172.216,43.846,158.508
C08053=1037.477,337.099,-124.774,172.211,43.843,158.507
C08054=1037.469,336.852,-124.738,172.205,43.841,158.506
C08055=1037.461,336.604,-124.702,172.200,43.839,158.505
C08056=1037.455,336.357,-124.665,172.196,43.837,158.504
C08057=1037.447,336.110,-124.629,172.191,43.834,158.504
C08058=1037.440,335.862,-124.593,172.186,43.832,158.503
C08059=1037.432,335.616,-124.557,172.180,43.830,158.502
C08060=1037.425,335.368,-124.521,172.175,43.828,158.501
C08061=1037.414,335.000,-124.467,172.168,43.825,158.499
C08062=1037.404,334.633,-124.414,172.160,43.821,158.498
C08063=1037.393,334.266,-124.360,172.153,43.818,158.496
C08064=1037.382,333.898,-124.306,172.145,43.815,158.495
C08065=1037.374,333.650,-124.271,172.140,43.813,158.494
C08066=1037.367,333.403,-124.236,172.135,43.810,158.493
C08067=1037.359,333.156,-124.199,172.130,43.808,158.492
C08068=1037.352,332.908,-124.164,172.124,43.806,158.491
C08069=1037.344,332.661,-124.128,172.120,43.803,158.490
C08070=1037.337,332.414,-124.092,172.115,43.802,158.489
C08071=1037.330,332.166,-124.057,172.110,43.800,158.488
C08072=1037.323,331.919,-124.021,172.105,43.797,158.488
C08073=1037.315,331.672,-123.985,172.100,43.795,158.487
C08074=1037.308,331.425,-123.949,172.095,43.793,158.486
C08075=1037.301,331.177,-123.913,172.090,43.791,158.485
C08076=1037.294,330.930,-123.878,172.085,43.789,158.484
C08077=1037.286,330.682,-123.842,172.080,43.787,158.483
C08078=1037.280,330.435,-123.807,172.075,43.785,158.482
C08079=1037.272,330.188,-123.770,172.070,43.783,158.481
C08080=1037.265,329.940,-123.735,172.065,43.780,158.480
C08081=1037.257,329.693,-123.699,172.061,43.779,158.479
C08082=1037.251,329.445,-123.664,172.056,43.776,158.478
C08083=1037.243,329.198,-123.628,172.051,43.774,158.477
C08084=1037.236,328.951,-123.593,172.046,43.773,158.477
C08085=1037.229,328.703,-123.558,172.041,43.770,158.476
C08086=1037.221,328.456,-123.522,172.036,43.768,158.475
C08087=1037.214,328.209,-123.487,172.031,43.766,158.474
C08088=1037.207,327.961,-123.451,172.026,43.765,158.473
C08089=1037.199,327.714,-123.417,172.021,43.762,158.472
C08090=1037.192,327.466,-123.381,172.017,43.761,158.471
C08091=1037.184,327.219,-123.346,172.012,43.758,158.470
C08092=1037.177,326.972,-123.311,172.007,43.757,158.470
C08093=1037.169,326.724,-123.276,172.002,43.755,158.469
C08094=1037.163,326.477,-123.241,171.998,43.753,158.468
C08095=1037.155,326.230,-123.206,171.993,43.751,158.467
C08096=1037.148,325.981,-123.171,171.988,43.749,158.466
C08097=1037.140,325.734,-123.136,171.983,43.747,158.465
C08098=1037.133,325.486,-123.101,171.979,43.745,158.465
C08099=1037.125,325.239,-123.066,171.974,43.744,158.464
C08100=1037.119,324.992,-123.031,171.969,43.741,158.463
C08101=1037.111,324.745,-122.996,171.964,43.740,158.462
C08102=1037.104,324.497,-122.961,171.960,43.738,158.461
C08103=1037.096,324.250,-122.926,171.955,43.736,158.461
C08104=1037.089,324.002,-122.891,171.950,43.734,158.460
C08105=1037.081,323.755,-122.856,171.946,43.732,158.459
C08106=1037.075,323.507,-122.821,171.941,43.730,158.458
C08107=1037.068,323.260,-122.786,171.936,43.729,158.457
C08108=1037.061,323.012,-122.752,171.931,43.727,158.456
C08109=1037.053,322.764,-122.717,171.927,43.725,158.455
C08110=1037.046,322.517,-122.682,171.922,43.723,158.455
C08111=1037.039,322.270,-122.647,171.917,43.721,158.454
C08112=1037.031,322.023,-122.613,171.913,43.720,158.453
C08113=1037.024,321.776,-122.578,171.908,43.717,158.452
C08114=1037.017,321.527,-122.543,171.903,43.716,158.451
C08115=1037.009,321.280,-122.509,171.899,43.714,158.451
C08116=1037.003,321.033,-122.474,171.894,43.712,158.450
C08117=1036.992,320.661,-122.421,171.887,43.709,158.449
C08118=1036.981,320.288,-122.369,171.880,43.707,158.447
C08119=1036.971,319.916,-122.317,171.873,43.704,158.446
C08120=1036.959,319.544,-122.265,171.866,43.701,158.445
C08121=1036.953,319.296,-122.231,171.862,43.699,158.444
C08122=1036.945,319.049,-122.196,171.857,43.698,158.443
C08123=1036.939,318.801,-122.161,171.853,43.696,158.443
C08124=1036.931,318.554,-122.127,171.848,43.694,158.442
C08125=1036.925,318.306,-122.092,171.843,43.693,158.441
C08126=1036.917,318.059,-122.058,171.839,43.691,158.440
C08127=1036.911,317.811,-122.023,171.834,43.689,158.439
C08128=1036.903,317.564,-121.990,171.830,43.687,158.439
C08129=1036.896,317.316,-121.955,171.825,43.686,158.438
C08130=1036.889,317.068,-121.921,171.820,43.684,158.437
C08131=1036.882,316.821,-121.886,171.816,43.682,158.436
C08132=1036.876,316.573,-121.852,171.811,43.680,158.436
C08133=1036.868,316.326,-121.818,171.807,43.678,158.435
C08134=1036.862,316.078,-121.783,171.802,43.677,158.434
C08135=1036.855,315.831,-121.749,171.799,43.675,158.433
C08136=1036.848,315.584,-121.714,171.794,43.673,158.432
C08137=1036.841,315.336,-121.680,171.790,43.672,158.432
C08138=1036.834,315.089,-121.646,171.785,43.670,158.431
C08139=1036.827,314.841,-121.611,171.781,43.669,158.430
C08140=1036.820,314.594,-121.577,171.776,43.667,158.429
C08141=1036.813,314.346,-121.543,171.772,43.665,158.429
C08142=1036.806,314.098,-121.509,171.767,43.663,158.428
C08143=1036.800,313.851,-121.474,171.763,43.661,158.427
C08144=1036.793,313.604,-121.441,171.758,43.660,158.426
C08145=1036.786,313.356,-121.407,171.755,43.659,158.426
C08146=1036.779,313.108,-121.372,171.750,43.657,158.425
C08147=1036.772,312.861,-121.338,171.746,43.655,158.424
C08148=1036.766,312.614,-121.304,171.741,43.653,158.423
C08149=1036.759,312.366,-121.270,171.737,43.651,158.423
C08150=1036.751,312.118,-121.236,171.732,43.650,158.422
C08151=1036.745,311.870,-121.202,171.728,43.649,158.421
C08152=1036.738,311.623,-121.168,171.723,43.647,158.420
C08153=1036.730,311.375,-121.134,171.719,43.646,158.420
C08154=1036.724,311.128,-121.101,171.714,43.644,158.419
C08155=1036.716,310.881,-121.067,171.711,43.642,158.418
C08156=1036.709,310.633,-121.034,171.706,43.641,158.418
C08157=1036.702,310.385,-121.000,171.702,43.639,158.417
C08158=1036.694,310.138,-120.966,171.697,43.638,158.416
C08159=1036.687,309.889,-120.933,171.693,43.636,158.416
C08160=1036.681,309.642,-120.899,171.689,43.635,158.415
C08161=1036.673,309.395,-120.866,171.685,43.633,158.414
C08162=1036.666,309.147,-120.832,171.680,43.632,158.414
C08163=1036.659,308.900,-120.798,171.676,43.631,158.413
C08164=1036.652,308.652,-120.766,171.672,43.629,158.412
C08165=1036.645,308.404,-120.732,171.667,43.628,158.412
C08166=1036.637,308.157,-120.699,171.664,43.626,158.411
C08167=1036.630,307.909,-120.666,171.659,43.625,158.410
C08168=1036.624,307.662,-120.632,171.655,43.623,158.409
C08169=1036.616,307.414,-120.598,171.650,43.622,158.409
C08170=1036.609,307.166,-120.564,171.646,43.621,158.408
C08171=1036.602,306.918,-120.531,171.642,43.619,158.407
C08172=1036.595,306.671,-120.498,171.638,43.618,158.407
C08173=1036.585,306.304,-120.449,171.632,43.616,158.406
C08174=1036.574,305.936,-120.399,171.625,43.614,158.405
C08175=1036.563,305.569,-120.350,171.619,43.612,158.404
C08176=1036.553,305.201,-120.301,171.613,43.610,158.403
C08177=1036.547,304.954,-120.268,171.608,43.608,158.402
C08178=1036.540,304.706,-120.234,171.604,43.607,158.401
C08179=1036.533,304.459,-120.202,171.601,43.605,158.401
C08180=1036.525,304.211,-120.168,171.596,43.604,158.400
C08181=1036.518,303.963,-120.135,171.592,43.602,158.399
C08182=1036.512,303.716,-120.101,171.587,43.601,158.399
C08183=1036.505,303.468,-120.068,171.584,43.600,158.398
C08184=1036.498,303.221,-120.035,171.580,43.598,158.397
C08185=1036.491,302.973,-120.002,171.575,43.597,158.397
C08186=1036.484,302.725,-119.970,171.571,43.596,158.396
C08187=1036.477,302.477,-119.936,171.568,43.595,158.396
C08188=1036.470,302.230,-119.904,171.563,43.593,158.395
C08189=1036.463,301.982,-119.871,171.559,43.592,158.394
C08190=1036.457,301.735,-119.837,171.555,43.590,158.394
C08191=1036.450,301.487,-119.804,171.551,43.589,158.393
C08192=1036.444,301.239,-119.771,171.547,43.587,158.392
C08193=1036.436,300.992,-119.738,171.543,43.586,158.392
C08194=1036.429,300.744,-119.705,171.538,43.585,158.391
C08195=1036.422,300.496,-119.672,171.534,43.584,158.390
C08196=1036.416,300.248,-119.639,171.531,43.582,158.390
C08197=1036.408,300.001,-119.606,171.526,43.581,158.389
C08198=1036.402,299.753,-119.573,171.522,43.579,158.388
C08199=1036.395,299.505,-119.540,171.518,43.578,158.388
C08200=1036.389,299.257,-119.508,171.515,43.577,158.387
C08201=1036.382,299.010,-119.475,171.510,43.576,158.387
C08202=1036.374,298.762,-119.442,171.506,43.574,158.386
C08203=1036.368,298.515,-119.409,171.502,43.573,158.385
C08204=1036.361,298.266,-119.376,171.499,43.571,158.385
C08205=1036.354,298.019,-119.344,171.494,43.570,158.384
C08206=1036.348,297.772,-119.311,171.490,43.569,158.384
C08207=1036.341,297.523,-119.278,171.486,43.568,158.383
C08208=1036.335,297.276,-119.245,171.483,43.567,158.382
C08209=1036.328,297.028,-119.213,171.478,43.565,158.382
C08210=1036.321,296.780,-119.180,171.474,43.564,158.381
C08211=1036.315,296.532,-119.147,171.470,43.562,158.380
C08212=1036.308,296.285,-119.114,171.467,43.561,158.380
C08213=1036.301,296.037,-119.082,171.462,43.560,158.379
C08214=1036.294,295.789,-119.049,171.458,43.559,158.379
C08215=1036.288,295.542,-119.016,171.455,43.557,158.378
C08216=1036.280,295.294,-118.984,171.451,43.556,158.377
C08217=1036.274,295.046,-118.951,171.447,43.555,158.377
C08218=1036.268,294.799,-118.918,171.442,43.554,158.376
C08219=1036.260,294.551,-118.886,171.439,43.552,158.376
C08220=1036.253,294.303,-118.854,171.435,43.551,158.375
C08221=1036.247,294.055,-118.822,171.431,43.550,158.374
C08222=1036.240,293.807,-118.789,171.427,43.549,158.374
C08223=1036.233,293.559,-118.756,171.423,43.548,158.373
C08224=1036.226,293.312,-118.724,171.419,43.547,158.373
C08225=1036.220,293.064,-118.692,171.416,43.546,158.372
C08226=1036.213,292.816,-118.660,171.412,43.544,158.372
C08227=1036.206,292.569,-118.627,171.407,43.543,158.371
C08228=1036.199,292.321,-118.596,171.404,43.542,158.370
C08229=1036.189,291.970,-118.550,171.399,43.540,158.369
C08230=1036.180,291.619,-118.505,171.393,43.539,158.369
C08231=1036.170,291.269,-118.459,171.388,43.537,158.368
C08232=1036.161,290.918,-118.414,171.382,43.535,158.367
C08233=1036.153,290.670,-118.381,171.378,43.535,158.367
C08234=1036.146,290.422,-118.350,171.375,43.533,158.366
C08235=1036.140,290.175,-118.317,171.371,43.532,158.365
C08236=1036.133,289.927,-118.286,171.366,43.531,158.365
C08237=1036.126,289.679,-118.253,171.363,43.530,158.364
C08238=1036.119,289.431,-118.222,171.359,43.529,158.364
C08239=1036.113,289.183,-118.189,171.355,43.528,158.363
C08240=1036.106,288.935,-118.158,171.352,43.527,158.363
C08241=1036.099,288.688,-118.125,171.348,43.526,158.362
C08242=1036.092,288.440,-118.094,171.344,43.525,158.362
C08243=1036.085,288.192,-118.062,171.340,43.524,158.361
C08244=1036.079,287.944,-118.029,171.336,43.523,158.361
C08245=1036.072,287.696,-117.998,171.333,43.522,158.360
C08246=1036.065,287.449,-117.966,171.329,43.520,158.359
C08247=1036.058,287.201,-117.934,171.325,43.520,158.359
C08248=1036.051,286.953,-117.903,171.322,43.518,158.358
C08249=1036.045,286.705,-117.871,171.317,43.517,158.358
C08250=1036.038,286.457,-117.838,171.314,43.517,158.357
C08251=1036.031,286.209,-117.807,171.310,43.515,158.357
C08252=1036.024,285.961,-117.776,171.306,43.515,158.356
C08253=1036.018,285.713,-117.744,171.303,43.513,158.356
C08254=1036.011,285.466,-117.712,171.299,43.513,158.355
C08255=1036.004,285.218,-117.681,171.295,43.511,158.355
C08256=1035.997,284.970,-117.649,171.292,43.511,158.354
C08257=1035.990,284.721,-117.617,171.287,43.510,158.354
C08258=1035.983,284.474,-117.586,171.284,43.509,158.353
C08259=1035.976,284.226,-117.554,171.280,43.508,158.353
C08260=1035.969,283.978,-117.524,171.277,43.507,158.352
C08261=1035.962,283.730,-117.492,171.273,43.506,158.351
C08262=1035.955,283.482,-117.461,171.269,43.505,158.351
C08263=1035.948,283.235,-117.429,171.266,43.504,158.350
C08264=1035.942,282.987,-117.397,171.262,43.503,158.350
C08265=1035.935,282.739,-117.366,171.259,43.502,158.349
C08266=1035.928,282.491,-117.334,171.255,43.501,158.349
C08267=1035.921,282.243,-117.303,171.251,43.500,158.348
C08268=1035.915,281.995,-117.271,171.248,43.499,158.348
C08269=1035.908,281.748,-117.240,171.243,43.498,158.347
C08270=1035.901,281.500,-117.209,171.240,43.497,158.347
C08271=1035.895,281.252,-117.177,171.236,43.496,158.346
C08272=1035.888,281.003,-117.146,171.233,43.495,158.346
C08273=1035.881,280.755,-117.115,171.229,43.494,158.345
C08274=1035.875,280.507,-117.084,171.225,43.493,158.345
C08275=1035.868,280.260,-117.052,171.222,43.492,158.344
C08276=1035.861,280.012,-117.021,171.218,43.491,158.344
C08277=1035.854,279.764,-116.989,171.215,43.491,158.343
C08278=1035.848,279.516,-116.958,171.211,43.489,158.343
C08279=1035.841,279.268,-116.926,171.208,43.489,158.342
C08280=1035.834,279.020,-116.895,171.204,43.487,158.342
C08281=1035.828,278.772,-116.864,171.200,43.487,158.341
C08282=1035.821,278.524,-116.833,171.197,43.486,158.341
C08283=1035.814,278.276,-116.802,171.193,43.485,158.340
C08284=1035.808,278.029,-116.771,171.190,43.484,158.340
C08285=1035.798,277.689,-116.729,171.185,43.483,158.339
C08286=1035.789,277.351,-116.686,171.180,43.482,158.339
C08287=1035.780,277.012,-116.644,171.175,43.480,158.338
C08288=1035.770,276.673,-116.602,171.171,43.479,158.337
C08289=1035.764,276.426,-116.570,171.167,43.478,158.337
C08290=1035.757,276.177,-116.540,171.164,43.478,158.336
C08291=1035.750,275.929,-116.509,171.160,43.477,158.336
C08292=1035.743,275.682,-116.477,171.157,43.476,158.335
C08293=1035.737,275.434,-116.447,171.153,43.475,158.335
C08294=1035.730,275.186,-116.416,171.150,43.474,158.334
C08295=1035.723,274.938,-116.385,171.146,43.474,158.334
C08296=1035.717,274.690,-116.354,171.142,43.472,158.333
C08297=1035.710,274.441,-116.323,171.139,43.472,158.333
C08298=1035.703,274.194,-116.293,171.135,43.471,158.333
C08299=1035.697,273.946,-116.262,171.132,43.470,158.332
C08300=1035.689,273.698,-116.231,171.128,43.469,158.332
C08301=1035.683,273.450,-116.201,171.125,43.468,158.331
C08302=1035.676,273.202,-116.169,171.121,43.468,158.331
C08303=1035.669,272.954,-116.139,171.118,43.467,158.330
C08304=1035.662,272.706,-116.108,171.114,43.466,158.330
C08305=1035.657,272.458,-116.077,171.111,43.466,158.329
C08306=1035.649,272.210,-116.047,171.107,43.464,158.329
C08307=1035.643,271.962,-116.016,171.104,43.464,158.328
C08308=1035.636,271.714,-115.986,171.100,43.463,158.328
C08309=1035.629,271.466,-115.954,171.097,43.462,158.328
C08310=1035.623,271.218,-115.924,171.093,43.462,158.327
C08311=1035.616,270.970,-115.894,171.090,43.461,158.327
C08312=1035.609,270.721,-115.863,171.086,43.460,158.326
C08313=1035.602,270.473,-115.832,171.084,43.459,158.326
C08314=1035.596,270.226,-115.802,171.080,43.458,158.325
C08315=1035.589,269.977,-115.772,171.077,43.457,158.325
C08316=1035.582,269.729,-115.742,171.073,43.457,158.324
C08317=1035.575,269.481,-115.710,171.070,43.456,158.324
C08318=1035.569,269.234,-115.680,171.066,43.455,158.324
C08319=1035.562,268.985,-115.650,171.063,43.455,158.323
C08320=1035.555,268.737,-115.620,171.059,43.454,158.323
C08321=1035.549,268.489,-115.589,171.056,43.453,158.322
C08322=1035.542,268.242,-115.558,171.052,43.453,158.322
C08323=1035.535,267.993,-115.528,171.049,43.452,158.321
C08324=1035.528,267.745,-115.497,171.046,43.451,158.321
C08325=1035.522,267.497,-115.468,171.043,43.450,158.321
C08326=1035.515,267.249,-115.437,171.040,43.450,158.320
C08327=1035.508,267.001,-115.407,171.036,43.449,158.320
C08328=1035.502,266.753,-115.377,171.033,43.448,158.319
C08329=1035.495,266.505,-115.346,171.029,43.448,158.319
C08330=1035.488,266.256,-115.316,171.026,43.447,158.318
C08331=1035.481,266.009,-115.287,171.022,43.446,158.318
C08332=1035.475,265.760,-115.256,171.019,43.445,158.318
C08333=1035.468,265.512,-115.226,171.016,43.445,158.317
C08334=1035.461,265.265,-115.196,171.013,43.444,158.317
C08335=1035.455,265.016,-115.165,171.009,43.443,158.316
C08336=1035.448,264.768,-115.135,171.006,43.442,158.316
C08337=1035.441,264.520,-115.105,171.002,43.442,158.315
C08338=1035.434,264.272,-115.075,170.999,43.441,158.315
C08339=1035.427,264.024,-115.045,170.995,43.440,158.315
C08340=1035.421,263.776,-115.015,170.993,43.440,158.314
C08341=1035.412,263.442,-114.974,170.988,43.439,158.314
C08342=1035.403,263.108,-114.934,170.984,43.438,158.313
C08343=1035.394,262.774,-114.893,170.979,43.437,158.313
C08344=1035.385,262.440,-114.853,170.975,43.436,158.312
C08345=1035.378,262.191,-114.823,170.971,43.436,158.312
C08346=1035.372,261.944,-114.793,170.969,43.435,158.311
C08347=1035.365,261.695,-114.764,170.965,43.434,158.311
C08348=1035.358,261.447,-114.734,170.962,43.434,158.310
C08349=1035.351,261.199,-114.704,170.958,43.433,158.310
C08350=1035.344,260.950,-114.674,170.955,43.433,158.310
C08351=1035.338,260.703,-114.645,170.951,43.432,158.309
C08352=1035.330,260.455,-114.614,170.949,43.432,158.309
C08353=1035.324,260.207,-114.585,170.946,43.431,158.308
C08354=1035.317,259.958,-114.555,170.942,43.430,158.308
C08355=1035.310,259.710,-114.526,170.939,43.430,158.308
C08356=1035.303,259.462,-114.497,170.936,43.429,158.307
C08357=1035.296,259.214,-114.467,170.932,43.429,158.307
C08358=1035.290,258.966,-114.438,170.930,43.429,158.307
C08359=1035.282,258.718,-114.407,170.926,43.428,158.306
C08360=1035.276,258.469,-114.378,170.923,43.427,158.306
C08361=1035.269,258.221,-114.348,170.919,43.426,158.305
C08362=1035.262,257.973,-114.319,170.916,43.426,158.305
C08363=1035.256,257.725,-114.289,170.913,43.426,158.305
C08364=1035.249,257.476,-114.260,170.910,43.425,158.304
C08365=1035.241,257.229,-114.231,170.907,43.425,158.304
C08366=1035.235,256.980,-114.201,170.903,43.424,158.304
C08367=1035.228,256.732,-114.172,170.900,43.423,158.303
C08368=1035.221,256.484,-114.142,170.897,43.423,158.303
C08369=1035.215,256.236,-114.113,170.894,43.422,158.302
C08370=1035.208,255.988,-114.083,170.891,43.422,158.302
C08371=1035.202,255.739,-114.054,170.888,43.422,158.302
C08372=1035.194,255.491,-114.024,170.884,43.421,158.301
C08373=1035.187,255.243,-113.995,170.882,43.420,158.301
C08374=1035.181,254.995,-113.966,170.878,43.420,158.301
C08375=1035.174,254.747,-113.936,170.875,43.419,158.300
C08376=1035.167,254.498,-113.907,170.871,43.419,158.300
C08377=1035.161,254.250,-113.878,170.869,43.418,158.300
C08378=1035.154,254.003,-113.848,170.866,43.418,158.299
C08379=1035.147,253.754,-113.818,170.862,43.417,158.299
C08380=1035.140,253.506,-113.790,170.859,43.417,158.298
C08381=1035.133,253.258,-113.760,170.857,43.416,158.298
C08382=1035.127,253.010,-113.731,170.853,43.415,158.298
C08383=1035.121,252.761,-113.702,170.850,43.415,158.297
C08384=1035.114,252.513,-113.672,170.846,43.414,158.297
C08385=1035.107,252.265,-113.643,170.844,43.414,158.297
C08386=1035.100,252.017,-113.614,170.841,43.414,158.296
C08387=1035.094,251.768,-113.585,170.837,43.413,158.296
C08388=1035.087,251.520,-113.556,170.834,43.413,158.295
C08389=1035.080,251.271,-113.526,170.831,43.412,158.295
C08390=1035.074,251.024,-113.497,170.828,43.411,158.295
C08391=1035.068,250.776,-113.468,170.825,43.411,158.294
C08392=1035.061,250.527,-113.438,170.822,43.410,158.294
C08393=1035.054,250.279,-113.410,170.819,43.410,158.294
C08394=1035.048,250.031,-113.381,170.815,43.409,158.293
C08395=1035.041,249.782,-113.351,170.813,43.409,158.293
C08396=1035.034,249.535,-113.321,170.810,43.408,158.293
C08397=1035.025,249.199,-113.282,170.805,43.408,158.292
C08398=1035.016,248.863,-113.244,170.802,43.407,158.292
C08399=1035.007,248.528,-113.204,170.797,43.406,158.291
C08400=1034.999,248.193,-113.165,170.794,43.405,158.291
C08401=1034.993,247.944,-113.135,170.790,43.405,158.290
C08402=1034.985,247.696,-113.107,170.787,43.405,158.290
C08403=1034.979,247.448,-113.078,170.784,43.404,158.290
C08404=1034.972,247.200,-113.049,170.781,43.404,158.289
C08405=1034.966,246.951,-113.020,170.778,43.403,158.289
C08406=1034.959,246.703,-112.990,170.775,43.403,158.289
C08407=1034.953,246.455,-112.961,170.772,43.402,158.288
C08408=1034.946,246.207,-112.933,170.769,43.401,158.288
C08409=1034.940,245.959,-112.904,170.766,43.401,158.288
C08410=1034.934,245.710,-112.875,170.763,43.400,158.287
C08411=1034.927,245.462,-112.845,170.761,43.400,158.287
C08412=1034.921,245.213,-112.816,170.757,43.399,158.286
C08413=1034.914,244.966,-112.788,170.754,43.399,158.286
C08414=1034.907,244.718,-112.759,170.751,43.398,158.286
C08415=1034.901,244.469,-112.730,170.748,43.398,158.285
C08416=1034.893,244.221,-112.701,170.745,43.398,158.285
C08417=1034.887,243.973,-112.672,170.742,43.397,158.285
C08418=1034.881,243.724,-112.644,170.739,43.397,158.284
C08419=1034.874,243.476,-112.615,170.737,43.396,158.284
C08420=1034.867,243.228,-112.586,170.733,43.396,158.284
C08421=1034.860,242.980,-112.557,170.730,43.396,158.283
C08422=1034.855,242.731,-112.529,170.728,43.395,158.283
C08423=1034.848,242.483,-112.500,170.724,43.395,158.283
C08424=1034.841,242.235,-112.471,170.721,43.394,158.282
C08425=1034.834,241.986,-112.443,170.719,43.394,158.282
C08426=1034.828,241.738,-112.414,170.715,43.393,158.282
C08427=1034.821,241.490,-112.386,170.713,43.393,158.281
C08428=1034.815,241.242,-112.357,170.710,43.393,158.281
C08429=1034.808,240.993,-112.329,170.706,43.392,158.281
C08430=1034.802,240.745,-112.300,170.704,43.392,158.280
C08431=1034.795,240.497,-112.271,170.700,43.391,158.280
C08432=1034.788,240.248,-112.243,170.698,43.391,158.280
C08433=1034.781,240.000,-112.214,170.695,43.391,158.280
C08434=1034.774,239.752,-112.186,170.691,43.390,158.279
C08435=1034.768,239.503,-112.158,170.689,43.390,158.279
C08436=1034.761,239.256,-112.129,170.686,43.390,158.279
C08437=1034.754,239.006,-112.101,170.683,43.389,158.278
C08438=1034.747,238.759,-112.073,170.680,43.389,158.278
C08439=1034.741,238.510,-112.044,170.677,43.389,158.278
C08440=1034.734,238.262,-112.016,170.674,43.388,158.277
C08441=1034.727,238.014,-111.988,170.671,43.388,158.277
C08442=1034.721,237.765,-111.959,170.669,43.387,158.277
C08443=1034.714,237.517,-111.931,170.666,43.387,158.276
C08444=1034.707,237.269,-111.903,170.663,43.386,158.276
C08445=1034.700,237.020,-111.875,170.660,43.386,158.276
C08446=1034.694,236.771,-111.846,170.657,43.386,158.276
C08447=1034.687,236.523,-111.818,170.654,43.385,158.275
C08448=1034.680,236.275,-111.790,170.651,43.385,158.275
C08449=1034.673,236.027,-111.762,170.649,43.385,158.275
C08450=1034.668,235.778,-111.733,170.646,43.385,158.274
C08451=1034.661,235.530,-111.706,170.643,43.384,158.274
C08452=1034.654,235.282,-111.677,170.640,43.384,158.274
C08453=1034.645,234.940,-111.639,170.636,43.383,158.273
C08454=1034.636,234.599,-111.601,170.632,43.383,158.273
C08455=1034.626,234.258,-111.561,170.629,43.383,158.272
C08456=1034.617,233.916,-111.523,170.624,43.382,158.272
C08457=1034.610,233.668,-111.495,170.622,43.382,158.272
C08458=1034.604,233.419,-111.467,170.618,43.381,158.271
C08459=1034.597,233.172,-111.439,170.616,43.381,158.271
C08460=1034.591,232.923,-111.410,170.613,43.381,158.271
C08461=1034.584,232.674,-111.383,170.611,43.380,158.271
C08462=1034.577,232.427,-111.354,170.607,43.380,158.270
C08463=1034.570,232.178,-111.326,170.605,43.379,158.270
C08464=1034.564,231.929,-111.298,170.602,43.379,158.270
C08465=1034.558,231.681,-111.270,170.599,43.379,158.269
C08466=1034.551,231.433,-111.243,170.596,43.378,158.269
C08467=1034.544,231.185,-111.214,170.593,43.378,158.269
C08468=1034.537,230.936,-111.187,170.591,43.378,158.268
C08469=1034.531,230.688,-111.159,170.587,43.378,158.268
C08470=1034.524,230.439,-111.131,170.585,43.378,158.268
C08471=1034.517,230.191,-111.103,170.582,43.377,158.268
C08472=1034.511,229.942,-111.076,170.579,43.377,158.267
C08473=1034.504,229.694,-111.048,170.576,43.377,158.267
C08474=1034.498,229.446,-111.020,170.574,43.376,158.267
C08475=1034.491,229.198,-110.993,170.572,43.376,158.267
C08476=1034.484,228.950,-110.964,170.568,43.375,158.266
C08477=1034.478,228.701,-110.936,170.566,43.375,158.266
C08478=1034.472,228.453,-110.908,170.563,43.375,158.266
C08479=1034.465,228.204,-110.881,170.560,43.375,158.265
C08480=1034.458,227.956,-110.853,170.557,43.375,158.265
C08481=1034.451,227.708,-110.826,170.555,43.374,158.265
C08482=1034.444,227.459,-110.798,170.552,43.374,158.265
C08483=1034.437,227.211,-110.770,170.549,43.373,158.264
C08484=1034.431,226.962,-110.743,170.546,43.373,158.264
C08485=1034.424,226.713,-110.715,170.544,43.373,158.264
C08486=1034.418,226.465,-110.688,170.540,43.373,158.263
C08487=1034.410,226.217,-110.661,170.538,43.373,158.263
C08488=1034.404,225.968,-110.633,170.535,43.373,158.263
C08489=1034.397,225.720,-110.605,170.533,43.372,158.263
C08490=1034.390,225.472,-110.577,170.529,43.372,158.262
C08491=1034.383,225.223,-110.550,170.527,43.372,158.262
C08492=1034.377,224.975,-110.522,170.524,43.372,158.262
C08493=1034.370,224.727,-110.496,170.522,43.372,158.262
C08494=1034.364,224.478,-110.468,170.518,43.372,158.261
C08495=1034.357,224.230,-110.440,170.516,43.371,158.261
C08496=1034.350,223.981,-110.413,170.514,43.370,158.261
C08497=1034.344,223.733,-110.385,170.510,43.370,158.260
C08498=1034.336,223.484,-110.359,170.508,43.370,158.260
C08499=1034.330,223.236,-110.331,170.505,43.370,158.260
C08500=1034.324,222.988,-110.303,170.503,43.370,158.260
C08501=1034.317,222.740,-110.276,170.499,43.370,158.259
C08502=1034.310,222.491,-110.248,170.497,43.369,158.259
C08503=1034.303,222.242,-110.222,170.495,43.369,158.259
C08504=1034.297,221.994,-110.194,170.492,43.369,158.259
C08505=1034.290,221.745,-110.166,170.490,43.369,158.258
C08506=1034.284,221.497,-110.139,170.486,43.369,158.258
C08507=1034.277,221.249,-110.112,170.484,43.368,158.258
C08508=1034.270,221.000,-110.085,170.482,43.368,158.258
C08509=1034.261,220.651,-110.047,170.477,43.368,158.257
C08510=1034.252,220.303,-110.007,170.474,43.368,158.257
C08511=1034.243,219.953,-109.969,170.470,43.367,158.256
C08512=1034.233,219.604,-109.931,170.466,43.367,158.256
C08513=1034.226,219.356,-109.904,170.464,43.367,158.256
C08514=1034.220,219.108,-109.877,170.461,43.367,158.256
C08515=1034.213,218.860,-109.850,170.459,43.366,158.255
C08516=1034.206,218.611,-109.822,170.455,43.366,158.255
C08517=1034.199,218.363,-109.796,170.453,43.366,158.255
C08518=1034.192,218.114,-109.768,170.451,43.366,158.255
C08519=1034.186,217.866,-109.742,170.448,43.366,158.254
C08520=1034.179,217.618,-109.715,170.445,43.365,158.254
C08521=1034.172,217.369,-109.688,170.442,43.365,158.254
C08522=1034.165,217.120,-109.660,170.440,43.365,158.254
C08523=1034.159,216.871,-109.633,170.438,43.365,158.253
C08524=1034.152,216.624,-109.607,170.434,43.365,158.253
C08525=1034.146,216.375,-109.580,170.432,43.364,158.253
C08526=1034.139,216.126,-109.553,170.430,43.364,158.253
C08527=1034.132,215.878,-109.525,170.427,43.364,158.252
C08528=1034.125,215.630,-109.499,170.424,43.364,158.252
C08529=1034.119,215.381,-109.472,170.421,43.364,158.252
C08530=1034.112,215.132,-109.445,170.419,43.364,158.252
C08531=1034.105,214.885,-109.418,170.417,43.364,158.252
C08532=1034.098,214.636,-109.391,170.414,43.364,158.251
C08533=1034.092,214.387,-109.364,170.411,43.363,158.251
C08534=1034.085,214.139,-109.337,170.409,43.363,158.251
C08535=1034.079,213.890,-109.311,170.406,43.363,158.251
C08536=1034.072,213.642,-109.284,170.404,43.363,158.250
C08537=1034.065,213.393,-109.257,170.401,43.362,158.250
C08538=1034.058,213.145,-109.230,170.398,43.362,158.250
C08539=1034.052,212.896,-109.203,170.396,43.362,158.250
C08540=1034.045,212.648,-109.176,170.394,43.362,158.249
C08541=1034.039,212.400,-109.150,170.390,43.362,158.249
C08542=1034.032,212.151,-109.123,170.388,43.361,158.249
C08543=1034.025,211.902,-109.096,170.386,43.361,158.249
C08544=1034.019,211.654,-109.069,170.383,43.361,158.248
C08545=1034.012,211.405,-109.042,170.380,43.361,158.248
C08546=1034.005,211.157,-109.015,170.378,43.361,158.248
C08547=1033.998,210.909,-108.989,170.375,43.360,158.248
C08548=1033.992,210.660,-108.962,170.373,43.361,158.247
C08549=1033.985,210.411,-108.936,170.371,43.361,158.247
C08550=1033.978,210.163,-108.910,170.367,43.360,158.247
C08551=1033.972,209.915,-108.882,170.365,43.360,158.247
C08552=1033.964,209.666,-108.856,170.363,43.360,158.246
C08553=1033.958,209.418,-108.830,170.361,43.360,158.246
C08554=1033.952,209.169,-108.803,170.357,43.360,158.246
C08555=1033.944,208.920,-108.776,170.355,43.359,158.246
C08556=1033.938,208.672,-108.750,170.353,43.360,158.246
C08557=1033.932,208.423,-108.723,170.350,43.360,158.245
C08558=1033.925,208.175,-108.697,170.348,43.359,158.245
C08559=1033.918,207.927,-108.670,170.345,43.359,158.245
C08560=1033.911,207.678,-108.643,170.342,43.359,158.245
C08561=1033.905,207.430,-108.617,170.340,43.359,158.244
C08562=1033.898,207.181,-108.590,170.338,43.359,158.244
C08563=1033.891,206.932,-108.564,170.336,43.359,158.244
C08564=1033.884,206.684,-108.538,170.332,43.359,158.244
C08565=1033.875,206.341,-108.501,170.329,43.359,158.243
C08566=1033.865,205.998,-108.465,170.326,43.358,158.243
C08567=1033.855,205.655,-108.429,170.323,43.358,158.243
C08568=1033.846,205.311,-108.393,170.319,43.358,158.243
C08569=1033.821,204.262,-108.287,169.988,43.254,158.195
C08570=1033.814,204.013,-108.262,169.985,43.254,158.195
C08571=1033.808,203.765,-108.237,169.982,43.255,158.194
C08572=1033.802,203.515,-108.212,169.978,43.255,158.194
C08573=1033.797,203.267,-108.187,169.975,43.256,158.194
C08574=1033.790,203.019,-108.162,169.971,43.257,158.194
C08575=1033.784,202.770,-108.136,169.968,43.257,158.194
C08576=1033.778,202.521,-108.112,169.964,43.259,158.194
C08577=1033.772,202.272,-108.086,169.961,43.259,158.194
C08578=1033.766,202.024,-108.062,169.958,43.260,158.194
C08579=1033.760,201.775,-108.037,169.954,43.260,158.193
C08580=1033.754,201.527,-108.012,169.950,43.261,158.193
C08581=1033.747,201.278,-107.987,169.947,43.261,158.193
C08582=1033.742,201.029,-107.962,169.943,43.262,158.193
C08583=1033.736,200.781,-107.937,169.940,43.263,158.193
C08584=1033.730,200.531,-107.912,169.936,43.263,158.193
C08585=1033.723,200.283,-107.888,169.933,43.265,158.193
C08586=1033.717,200.034,-107.863,169.930,43.265,158.193
C08587=1033.711,199.786,-107.839,169.926,43.266,158.192
C08588=1033.705,199.537,-107.814,169.924,43.267,158.192
C08589=1033.698,199.288,-107.789,169.920,43.268,158.192
C08590=1033.692,199.039,-107.765,169.916,43.268,158.192
C08591=1033.685,198.791,-107.740,169.913,43.269,158.192
C08592=1033.680,198.542,-107.716,169.910,43.270,158.192
C08593=1033.673,198.293,-107.692,169.907,43.271,158.192
C08594=1033.667,198.044,-107.666,169.902,43.271,158.192
C08595=1033.660,197.795,-107.642,169.900,43.272,158.192
C08596=1033.655,197.547,-107.618,169.897,43.273,158.191
C08597=1033.648,197.299,-107.593,169.893,43.274,158.191
C08598=1033.642,197.049,-107.569,169.890,43.275,158.191
C08599=1033.637,196.801,-107.544,169.886,43.276,158.191
C08600=1033.630,196.552,-107.520,169.883,43.276,158.191
C08601=1033.624,196.303,-107.495,169.880,43.277,158.191
C08602=1033.618,196.055,-107.471,169.876,43.278,158.191
C08603=1033.612,195.806,-107.446,169.873,43.279,158.191
C08604=1033.605,195.557,-107.422,169.870,43.280,158.191
C08605=1033.600,195.308,-107.398,169.866,43.280,158.191
C08606=1033.593,195.060,-107.373,169.863,43.282,158.191
C08607=1033.587,194.811,-107.348,169.860,43.282,158.190
C08608=1033.581,194.563,-107.325,169.856,43.283,158.190
C08609=1033.575,194.313,-107.300,169.853,43.284,158.190
C08610=1033.568,194.065,-107.275,169.850,43.285,158.190
C08611=1033.563,193.816,-107.251,169.846,43.285,158.190
C08612=1033.556,193.567,-107.227,169.843,43.286,158.190
C08613=1033.550,193.318,-107.202,169.840,43.287,158.190
C08614=1033.544,193.070,-107.179,169.836,43.288,158.190
C08615=1033.538,192.820,-107.154,169.833,43.289,158.190
C08616=1033.532,192.573,-107.130,169.830,43.289,158.190
C08617=1033.525,192.324,-107.106,169.826,43.291,158.190
C08618=1033.520,192.075,-107.081,169.823,43.291,158.189
C08619=1033.514,191.826,-107.057,169.821,43.292,158.189
C08620=1033.508,191.577,-107.033,169.817,43.293,158.189
C08621=1033.502,191.329,-107.009,169.813,43.294,158.189
C08622=1033.496,191.079,-106.985,169.811,43.295,158.189
C08623=1033.490,190.831,-106.961,169.808,43.295,158.189
C08624=1033.483,190.583,-106.936,169.804,43.297,158.189
C08625=1033.477,190.334,-106.912,169.801,43.297,158.189
C08626=1033.471,190.085,-106.887,169.798,43.298,158.189
C08627=1033.465,189.837,-106.864,169.795,43.299,158.189
C08628=1033.460,189.587,-106.839,169.791,43.300,158.189
C08629=1033.454,189.339,-106.815,169.788,43.301,158.189
C08630=1033.446,189.054,-106.788,169.784,43.302,158.188
C08631=1033.440,188.771,-106.760,169.781,43.303,158.188
C08632=1033.433,188.487,-106.733,169.777,43.304,158.188
C08633=1033.426,188.203,-106.706,169.773,43.305,158.188
C08634=1033.420,187.954,-106.682,169.770,43.305,158.188
C08635=1033.415,187.706,-106.657,169.767,43.307,158.188
C08636=1033.408,187.457,-106.633,169.764,43.307,158.188
C08637=1033.403,187.208,-106.609,169.760,43.308,158.188
C08638=1033.397,186.960,-106.585,169.757,43.309,158.188
C08639=1033.391,186.710,-106.561,169.755,43.310,158.188
C08640=1033.385,186.462,-106.537,169.751,43.311,158.188
C08641=1033.379,186.213,-106.512,169.749,43.312,158.188
C08642=1033.373,185.965,-106.489,169.745,43.313,158.188
C08643=1033.367,185.715,-106.464,169.742,43.313,158.187
C08644=1033.361,185.466,-106.441,169.739,43.314,158.187
C08645=1033.355,185.218,-106.418,169.736,43.315,158.187
C08646=1033.349,184.969,-106.393,169.733,43.316,158.187
C08647=1033.343,184.721,-106.369,169.729,43.317,158.187
C08648=1033.337,184.471,-106.345,169.726,43.318,158.187
C08649=1033.331,184.223,-106.321,169.723,43.318,158.187
C08650=1033.326,183.974,-106.297,169.720,43.320,158.187
C08651=1033.320,183.725,-106.273,169.717,43.320,158.187
C08652=1033.313,183.476,-106.250,169.714,43.321,158.187
C08653=1033.308,183.228,-106.225,169.710,43.322,158.187
C08654=1033.302,182.978,-106.202,169.707,43.323,158.187
C08655=1033.296,182.730,-106.179,169.705,43.324,158.187
C08656=1033.289,182.481,-106.154,169.702,43.326,158.187
C08657=1033.283,182.232,-106.132,169.698,43.326,158.187
C08658=1033.276,181.983,-106.108,169.695,43.327,158.187
C08659=1033.270,181.735,-106.085,169.692,43.329,158.187
C08660=1033.264,181.486,-106.062,169.689,43.330,158.187
C08661=1033.258,181.237,-106.038,169.686,43.331,158.187
C08662=1033.252,180.988,-106.015,169.682,43.332,158.186
C08663=1033.246,180.739,-105.991,169.679,43.333,158.186
C08664=1033.240,180.491,-105.968,169.677,43.334,158.187
C08665=1033.233,180.242,-105.945,169.674,43.335,158.187
C08666=1033.226,179.993,-105.921,169.670,43.337,158.186
C08667=1033.221,179.744,-105.898,169.667,43.338,158.187
C08668=1033.214,179.495,-105.874,169.664,43.338,158.186
C08669=1033.208,179.246,-105.851,169.661,43.340,158.186
C08670=1033.202,178.998,-105.828,169.658,43.341,158.186
C08671=1033.196,178.748,-105.804,169.655,43.342,158.186
C08672=1033.190,178.500,-105.782,169.652,43.343,158.186
C08673=1033.183,178.251,-105.758,169.649,43.344,158.186
C08674=1033.177,178.002,-105.735,169.646,43.345,158.186
C08675=1033.171,177.754,-105.711,169.643,43.346,158.186
C08676=1033.165,177.505,-105.688,169.639,43.348,158.186
C08677=1033.159,177.255,-105.665,169.636,43.349,158.186
C08678=1033.152,177.007,-105.642,169.634,43.350,158.186
C08679=1033.147,176.758,-105.619,169.631,43.351,158.186
C08680=1033.140,176.509,-105.596,169.628,43.352,158.186
C08681=1033.134,176.260,-105.572,169.624,43.353,158.186
C08682=1033.128,176.011,-105.549,169.621,43.354,158.186
C08683=1033.122,175.763,-105.527,169.618,43.355,158.186
C08684=1033.115,175.514,-105.503,169.615,43.357,158.186
C08685=1033.110,175.265,-105.480,169.613,43.358,158.186
C08686=1033.104,175.016,-105.457,169.610,43.359,158.186
C08687=1033.098,174.767,-105.434,169.607,43.360,158.186
C08688=1033.092,174.518,-105.410,169.603,43.361,158.186
C08689=1033.085,174.270,-105.388,169.600,43.362,158.186
C08690=1033.079,174.021,-105.365,169.597,43.363,158.186
C08691=1033.074,173.772,-105.342,169.594,43.364,158.186
C08692=1033.067,173.523,-105.318,169.592,43.365,158.186
C08693=1033.061,173.274,-105.295,169.589,43.367,158.186
C08694=1033.054,172.990,-105.269,169.585,43.368,158.186
C08695=1033.047,172.706,-105.243,169.582,43.369,158.186
C08696=1033.041,172.422,-105.216,169.578,43.371,158.186
C08697=1033.034,172.137,-105.190,169.575,43.372,158.186
C08698=1033.027,171.888,-105.167,169.572,43.373,158.186
C08699=1033.021,171.639,-105.144,169.568,43.374,158.186
C08700=1033.015,171.391,-105.121,169.566,43.375,158.186
C08701=1033.009,171.142,-105.098,169.563,43.376,158.186
C08702=1033.004,170.893,-105.075,169.560,43.377,158.186
C08703=1032.998,170.644,-105.052,169.557,43.378,158.186
C08704=1032.991,170.395,-105.029,169.554,43.380,158.186
C08705=1032.985,170.146,-105.006,169.552,43.381,158.186
C08706=1032.979,169.897,-104.983,169.549,43.382,158.186
C08707=1032.974,169.648,-104.960,169.546,43.383,158.186
C08708=1032.968,169.399,-104.937,169.543,43.384,158.186
C08709=1032.961,169.151,-104.914,169.539,43.385,158.186
C08710=1032.955,168.902,-104.891,169.536,43.386,158.186
C08711=1032.950,168.653,-104.868,169.533,43.387,158.186
C08712=1032.943,168.404,-104.845,169.530,43.389,158.186
C08713=1032.937,168.155,-104.823,169.528,43.390,158.186
C08714=1032.931,167.906,-104.800,169.525,43.391,158.186
C08715=1032.925,167.657,-104.777,169.522,43.392,158.186
C08716=1032.920,167.408,-104.754,169.519,43.393,158.186
C08717=1032.914,167.160,-104.731,169.516,43.395,158.186
C08718=1032.907,166.911,-104.708,169.513,43.395,158.186
C08719=1032.902,166.662,-104.686,169.510,43.396,158.186
C08720=1032.896,166.413,-104.663,169.508,43.397,158.186
C08721=1032.890,166.164,-104.640,169.505,43.399,158.186
C08722=1032.884,165.916,-104.617,169.502,43.400,158.186
C08723=1032.878,165.666,-104.595,169.499,43.401,158.186
C08724=1032.873,165.417,-104.572,169.496,43.402,158.186
C08725=1032.867,165.168,-104.549,169.494,43.403,158.186
C08726=1032.861,164.920,-104.526,169.491,43.405,158.186
C08727=1032.855,164.671,-104.504,169.488,43.406,158.186
C08728=1032.849,164.422,-104.481,169.485,43.407,158.186
C08729=1032.843,164.173,-104.458,169.482,43.407,158.186
C08730=1032.837,163.924,-104.435,169.479,43.409,158.186
C08731=1032.831,163.676,-104.413,169.476,43.410,158.186
C08732=1032.826,163.426,-104.390,169.473,43.411,158.186
C08733=1032.820,163.177,-104.368,169.471,43.412,158.186
C08734=1032.814,162.928,-104.345,169.468,43.413,158.186
C08735=1032.808,162.680,-104.322,169.465,43.415,158.186
C08736=1032.802,162.431,-104.299,169.462,43.416,158.186
C08737=1032.796,162.182,-104.276,169.459,43.417,158.186
C08738=1032.791,161.932,-104.254,169.457,43.418,158.186
C08739=1032.784,161.684,-104.232,169.454,43.419,158.186
C08740=1032.779,161.435,-104.209,169.451,43.420,158.186
C08741=1032.773,161.186,-104.186,169.448,43.421,158.186
C08742=1032.767,160.937,-104.163,169.445,43.422,158.186
C08743=1032.761,160.688,-104.141,169.442,43.423,158.186
C08744=1032.755,160.439,-104.118,169.439,43.425,158.186
C08745=1032.749,160.190,-104.095,169.437,43.426,158.186
C08746=1032.743,159.942,-104.073,169.434,43.427,158.186
C08747=1032.738,159.692,-104.051,169.431,43.428,158.186
C08748=1032.731,159.443,-104.028,169.428,43.429,158.186
C08749=1032.726,159.194,-104.006,169.425,43.431,158.186
C08750=1032.719,158.945,-103.984,169.422,43.432,158.186
C08751=1032.714,158.697,-103.963,169.420,43.434,158.186
C08752=1032.708,158.448,-103.940,169.417,43.435,158.186
C08753=1032.701,158.199,-103.917,169.414,43.436,158.186
C08754=1032.695,157.950,-103.896,169.411,43.437,158.186
C08755=1032.690,157.701,-103.873,169.408,43.438,158.186
C08756=1032.683,157.452,-103.851,169.406,43.440,158.186
C08757=1032.677,157.204,-103.829,169.403,43.441,158.186
C08758=1032.670,156.918,-103.804,169.400,43.443,158.186
C08759=1032.663,156.634,-103.778,169.396,43.444,158.186
C08760=1032.657,156.349,-103.753,169.394,43.445,158.186
C08761=1032.650,156.064,-103.727,169.391,43.447,158.186
C08762=1032.644,155.815,-103.706,169.388,43.448,158.186
C08763=1032.637,155.567,-103.683,169.385,43.449,158.186
C08764=1032.632,155.317,-103.661,169.382,43.451,158.186
C08765=1032.625,155.069,-103.639,169.380,43.452,158.186
C08766=1032.619,154.819,-103.617,169.377,43.453,158.186
C08767=1032.614,154.570,-103.594,169.374,43.455,158.186
C08768=1032.607,154.321,-103.573,169.371,43.456,158.186
C08769=1032.601,154.072,-103.551,169.368,43.457,158.186
C08770=1032.595,153.824,-103.529,169.366,43.458,158.186
C08771=1032.590,153.575,-103.507,169.363,43.460,158.187
C08772=1032.583,153.326,-103.484,169.360,43.461,158.187
C08773=1032.577,153.077,-103.463,169.357,43.463,158.187
C08774=1032.571,152.828,-103.441,169.355,43.464,158.187
C08775=1032.565,152.578,-103.420,169.352,43.465,158.187
C08776=1032.558,152.330,-103.397,169.349,43.466,158.187
C08777=1032.554,152.081,-103.375,169.346,43.468,158.187
C08778=1032.548,151.832,-103.354,169.343,43.469,158.187
C08779=1032.541,151.583,-103.331,169.341,43.470,158.187
C08780=1032.535,151.334,-103.310,169.338,43.472,158.187
C08781=1032.529,151.085,-103.288,169.335,43.473,158.187
C08782=1032.523,150.836,-103.266,169.332,43.475,158.187
C08783=1032.517,150.588,-103.244,169.331,43.476,158.187
C08784=1032.511,150.338,-103.222,169.328,43.477,158.187
C08785=1032.505,150.089,-103.201,169.325,43.478,158.187
C08786=1032.499,149.840,-103.179,169.322,43.480,158.187
C08787=1032.492,149.591,-103.157,169.319,43.481,158.187
C08788=1032.487,149.343,-103.135,169.317,43.482,158.187
C08789=1032.481,149.094,-103.114,169.314,43.483,158.187
C08790=1032.475,148.844,-103.092,169.311,43.485,158.187
C08791=1032.468,148.595,-103.070,169.308,43.486,158.187
C08792=1032.463,148.346,-103.048,169.306,43.488,158.187
C08793=1032.457,148.098,-103.026,169.303,43.489,158.187
C08794=1032.451,147.848,-103.005,169.300,43.491,158.188
C08795=1032.445,147.599,-102.983,169.297,43.492,158.188
C08796=1032.439,147.350,-102.961,169.295,43.493,158.188
C08797=1032.433,147.102,-102.940,169.293,43.494,158.188
C08798=1032.427,146.852,-102.918,169.290,43.496,158.188
C08799=1032.421,146.603,-102.897,169.287,43.497,158.188
C08800=1032.415,146.354,-102.875,169.284,43.498,158.188
C08801=1032.408,146.105,-102.853,169.282,43.500,158.188
C08802=1032.403,145.856,-102.832,169.279,43.501,158.188
C08803=1032.397,145.607,-102.811,169.276,43.503,158.188
C08804=1032.390,145.358,-102.790,169.273,43.504,158.188
C08805=1032.384,145.109,-102.768,169.271,43.506,158.188
C08806=1032.378,144.860,-102.747,169.268,43.507,158.188
C08807=1032.372,144.611,-102.725,169.265,43.509,158.188
C08808=1032.366,144.362,-102.703,169.262,43.510,158.188
C08809=1032.360,144.113,-102.682,169.261,43.511,158.188
C08810=1032.354,143.864,-102.660,169.258,43.513,158.189
C08811=1032.348,143.615,-102.639,169.255,43.514,158.189
C08812=1032.341,143.366,-102.618,169.252,43.516,158.189
C08813=1032.335,143.118,-102.597,169.250,43.517,158.189
C08814=1032.329,142.869,-102.575,169.247,43.518,158.189
C08815=1032.323,142.619,-102.553,169.244,43.520,158.189
C08816=1032.317,142.371,-102.532,169.241,43.521,158.189
C08817=1032.312,142.121,-102.511,169.239,43.522,158.189
C08818=1032.305,141.872,-102.489,169.237,43.524,158.189
C08819=1032.299,141.623,-102.468,169.234,43.525,158.189
C08820=1032.293,141.374,-102.447,169.231,43.526,158.189
C08821=1032.287,141.125,-102.425,169.229,43.528,158.189
C08822=1032.280,140.840,-102.401,169.226,43.530,158.189
C08823=1032.273,140.555,-102.377,169.222,43.532,158.189
C08824=1032.267,140.270,-102.352,169.219,43.533,158.189
C08825=1032.259,139.985,-102.328,169.217,43.535,158.189
C08826=1032.254,139.736,-102.306,169.214,43.536,158.189
C08827=1032.248,139.487,-102.285,169.211,43.537,158.189
C08828=1032.242,139.237,-102.264,169.209,43.539,158.190
C08829=1032.235,138.989,-102.243,169.206,43.540,158.190
C08830=1032.229,138.740,-102.221,169.203,43.541,158.190
C08831=1032.224,138.491,-102.201,169.201,43.543,158.190
C08832=1032.218,138.242,-102.179,169.198,43.544,158.190
C08833=1032.211,137.993,-102.158,169.196,43.546,158.190
C08834=1032.205,137.744,-102.137,169.193,43.547,158.190
C08835=1032.200,137.494,-102.116,169.190,43.549,158.190
C08836=1032.193,137.245,-102.095,169.188,43.550,158.190
C08837=1032.187,136.997,-102.074,169.185,43.551,158.190
C08838=1032.181,136.747,-102.053,169.182,43.553,158.190
C08839=1032.175,136.499,-102.032,169.180,43.554,158.190
C08840=1032.169,136.250,-102.010,169.178,43.556,158.191
C08841=1032.163,136.000,-101.990,169.175,43.557,158.191
C08842=1032.157,135.752,-101.969,169.172,43.559,158.191
C08843=1032.151,135.502,-101.948,169.169,43.560,158.191
C08844=1032.145,135.253,-101.927,169.167,43.562,158.191
C08845=1032.138,135.004,-101.906,169.164,43.563,158.191
C08846=1032.132,134.755,-101.885,169.162,43.564,158.191
C08847=1032.126,134.506,-101.864,169.160,43.566,158.191
C08848=1032.120,134.257,-101.843,169.157,43.568,158.191
C08849=1032.115,134.008,-101.822,169.154,43.569,158.191
C08850=1032.108,133.759,-101.801,169.151,43.571,158.191
C08851=1032.103,133.510,-101.780,169.149,43.572,158.191
C08852=1032.096,133.261,-101.759,169.147,43.573,158.191
C08853=1032.090,133.011,-101.738,169.144,43.575,158.192
C08854=1032.084,132.763,-101.717,169.141,43.576,158.192
C08855=1032.078,132.513,-101.697,169.139,43.578,158.192
C08856=1032.072,132.265,-101.675,169.136,43.580,158.192
C08857=1032.066,132.015,-101.655,169.133,43.581,158.192
C08858=1032.060,131.767,-101.634,169.132,43.582,158.192
C08859=1032.054,131.517,-101.613,169.129,43.584,158.192
C08860=1032.048,131.269,-101.592,169.126,43.585,158.192
C08861=1032.042,131.019,-101.571,169.123,43.587,158.192
C08862=1032.036,130.771,-101.551,169.120,43.588,158.192
C08863=1032.030,130.521,-101.530,169.118,43.590,158.192
C08864=1032.024,130.272,-101.510,169.116,43.591,158.192
C08865=1032.017,130.023,-101.489,169.113,43.593,158.192
C08866=1032.012,129.774,-101.468,169.111,43.594,158.193
C08867=1032.005,129.525,-101.448,169.108,43.596,158.193
C08868=1031.998,129.276,-101.427,169.105,43.598,158.193
C08869=1031.992,129.027,-101.407,169.103,43.599,158.193
C08870=1031.986,128.777,-101.386,169.100,43.601,158.193
C08871=1031.980,128.529,-101.365,169.098,43.602,158.193
C08872=1031.973,128.279,-101.345,169.096,43.603,158.193
C08873=1031.968,128.030,-101.324,169.093,43.605,158.193
C08874=1031.962,127.781,-101.304,169.090,43.607,158.193
C08875=1031.955,127.533,-101.283,169.087,43.608,158.193
C08876=1031.949,127.283,-101.263,169.085,43.610,158.193
C08877=1031.943,127.034,-101.242,169.082,43.611,158.193
C08878=1031.937,126.784,-101.222,169.080,43.613,158.194
C08879=1031.931,126.536,-101.201,169.078,43.615,158.194
C08880=1031.924,126.287,-101.181,169.075,43.616,158.194
C08881=1031.919,126.038,-101.161,169.072,43.618,158.194
C08882=1031.912,125.788,-101.140,169.070,43.619,158.194
C08883=1031.906,125.540,-101.120,169.067,43.621,158.194
C08884=1031.900,125.291,-101.100,169.065,43.622,158.194
C08885=1031.894,125.041,-101.079,169.063,43.624,158.194
C08886=1031.886,124.756,-101.056,169.060,43.626,158.194
C08887=1031.880,124.471,-101.032,169.056,43.628,158.195
C08888=1031.873,124.186,-101.009,169.053,43.629,158.195
C08889=1031.866,123.901,-100.985,169.051,43.631,158.195
C08890=1031.860,123.652,-100.965,169.048,43.633,158.195
C08891=1031.853,123.402,-100.945,169.045,43.634,158.195
C08892=1031.847,123.154,-100.925,169.043,43.636,158.195
C08893=1031.841,122.904,-100.904,169.041,43.638,158.195
C08894=1031.835,122.655,-100.884,169.038,43.639,158.195
C08895=1031.829,122.406,-100.864,169.036,43.641,158.195
C08896=1031.822,122.157,-100.843,169.033,43.642,158.195
C08897=1031.817,121.908,-100.822,169.030,43.644,158.196
C08898=1031.811,121.659,-100.802,169.029,43.645,158.196
C08899=1031.805,121.410,-100.782,169.026,43.647,158.196
C08900=1031.799,121.161,-100.762,169.023,43.648,158.196
C08901=1031.793,120.911,-100.741,169.020,43.650,158.196
C08902=1031.787,120.662,-100.721,169.019,43.651,158.196
C08903=1031.781,120.414,-100.701,169.016,43.653,158.196
C08904=1031.774,120.164,-100.681,169.013,43.654,158.196
C08905=1031.769,119.915,-100.660,169.011,43.656,158.196
C08906=1031.763,119.666,-100.640,169.008,43.658,158.196
C08907=1031.756,119.417,-100.620,169.006,43.659,158.196
C08908=1031.750,119.168,-100.600,169.004,43.660,158.197
C08909=1031.744,118.919,-100.580,169.001,43.662,158.197
C08910=1031.738,118.669,-100.559,168.998,43.663,158.197
C08911=1031.732,118.420,-100.539,168.996,43.665,158.197
C08912=1031.726,118.171,-100.519,168.994,43.666,158.197
C08913=1031.720,117.922,-100.499,168.991,43.668,158.197
C08914=1031.715,117.673,-100.479,168.988,43.669,158.197
C08915=1031.709,117.424,-100.459,168.987,43.671,158.197
C08916=1031.702,117.174,-100.438,168.984,43.672,158.197
C08917=1031.696,116.926,-100.418,168.981,43.674,158.197
C08918=1031.690,116.677,-100.398,168.978,43.675,158.197
C08919=1031.685,116.428,-100.378,168.977,43.677,158.198
C08920=1031.678,116.178,-100.357,168.974,43.678,158.198
C08921=1031.672,115.929,-100.337,168.971,43.680,158.198
C08922=1031.666,115.681,-100.318,168.969,43.681,158.198
C08923=1031.661,115.431,-100.297,168.967,43.683,158.198
C08924=1031.654,115.182,-100.277,168.964,43.684,158.198
C08925=1031.649,114.933,-100.257,168.962,43.686,158.198
C08926=1031.643,114.684,-100.237,168.960,43.687,158.198
C08927=1031.637,114.435,-100.217,168.957,43.689,158.198
C08928=1031.631,114.185,-100.197,168.954,43.690,158.198
C08929=1031.625,113.936,-100.177,168.952,43.692,158.198
C08930=1031.619,113.687,-100.157,168.950,43.693,158.198
C08931=1031.613,113.439,-100.137,168.947,43.695,158.199
C08932=1031.607,113.189,-100.117,168.944,43.696,158.199
C08933=1031.601,112.940,-100.097,168.942,43.698,158.199
C08934=1031.595,112.691,-100.077,168.940,43.699,158.199
C08935=1031.588,112.441,-100.057,168.937,43.701,158.199
C08936=1031.582,112.192,-100.038,168.935,43.703,158.199
C08937=1031.576,111.943,-100.018,168.932,43.704,158.199
C08938=1031.570,111.694,-99.998,168.930,43.706,158.199
C08939=1031.564,111.446,-99.978,168.928,43.708,158.199
C08940=1031.558,111.195,-99.958,168.925,43.709,158.199
C08941=1031.552,110.947,-99.938,168.922,43.711,158.200
C08942=1031.546,110.698,-99.918,168.921,43.712,158.200
C08943=1031.540,110.448,-99.899,168.918,43.714,158.200
C08944=1031.534,110.199,-99.879,168.915,43.715,158.200
C08945=1031.528,109.950,-99.859,168.913,43.717,158.200
C08946=1031.521,109.701,-99.840,168.911,43.718,158.200
C08947=1031.515,109.452,-99.820,168.908,43.720,158.200
C08948=1031.509,109.202,-99.800,168.906,43.722,158.200
C08949=1031.503,108.953,-99.780,168.903,43.723,158.200
C08950=1031.496,108.668,-99.758,168.900,43.725,158.200
C08951=1031.489,108.382,-99.736,168.898,43.727,158.201
C08952=1031.481,108.097,-99.713,168.895,43.729,158.201
C08953=1031.474,107.812,-99.691,168.892,43.731,158.201
C08954=1031.468,107.563,-99.672,168.890,43.733,158.201
C08955=1031.462,107.314,-99.652,168.887,43.735,158.201
C08956=1031.456,107.064,-99.632,168.884,43.736,158.201
C08957=1031.450,106.815,-99.612,168.883,43.737,158.201
C08958=1031.444,106.566,-99.594,168.880,43.739,158.202
C08959=1031.438,106.317,-99.574,168.877,43.741,158.202
C08960=1031.432,106.068,-99.554,168.875,43.742,158.202
C08961=1031.426,105.819,-99.535,168.873,43.744,158.202
C08962=1031.419,105.569,-99.516,168.870,43.745,158.202
C08963=1031.413,105.320,-99.496,168.868,43.747,158.202
C08964=1031.407,105.071,-99.476,168.865,43.749,158.202
C08965=1031.401,104.822,-99.456,168.863,43.750,158.202
C08966=1031.395,104.573,-99.438,168.861,43.752,158.202
C08967=1031.389,104.324,-99.418,168.858,43.754,158.202
C08968=1031.383,104.074,-99.398,168.855,43.756,158.203
C08969=1031.377,103.825,-99.378,168.854,43.757,158.203
C08970=1031.370,103.576,-99.360,168.851,43.759,158.203
C08971=1031.364,103.327,-99.340,168.848,43.761,158.203
C08972=1031.359,103.078,-99.320,168.847,43.762,158.203
C08973=1031.352,102.829,-99.302,168.844,43.763,158.203
C08974=1031.346,102.580,-99.282,168.841,43.765,158.203
C08975=1031.340,102.330,-99.262,168.839,43.767,158.203
C08976=1031.334,102.082,-99.243,168.837,43.768,158.203
C08977=1031.328,101.833,-99.224,168.834,43.769,158.203
C08978=1031.322,101.582,-99.204,168.831,43.771,158.204
C08979=1031.316,101.334,-99.184,168.830,43.773,158.204
C08980=1031.310,101.084,-99.165,168.827,43.774,158.204
C08981=1031.304,100.835,-99.146,168.824,43.776,158.204
C08982=1031.298,100.586,-99.126,168.822,43.778,158.204
C08983=1031.292,100.337,-99.107,168.820,43.779,158.204
C08984=1031.286,100.087,-99.088,168.817,43.781,158.204
C08985=1031.280,99.839,-99.069,168.815,43.783,158.204
C08986=1031.274,99.589,-99.049,168.813,43.784,158.204
C08987=1031.267,99.340,-99.031,168.810,43.786,158.205
C08988=1031.262,99.091,-99.011,168.808,43.788,158.205
C08989=1031.254,98.842,-98.992,168.805,43.789,158.205
C08990=1031.248,98.593,-98.973,168.803,43.790,158.205
C08991=1031.242,98.343,-98.954,168.801,43.792,158.205
C08992=1031.236,98.094,-98.935,168.798,43.794,158.205
C08993=1031.230,97.845,-98.916,168.796,43.796,158.205
C08994=1031.223,97.596,-98.897,168.794,43.798,158.206
C08995=1031.218,97.347,-98.877,168.791,43.799,158.206
